LIN {X 0,Y 334.107,Z 246.869,A -85,B 0,C 180,E1 -14402.411,E2 -14402.411} C_VEL
LIN {X 0,Y 334.001,Z 246.88,A -85,B 0,C 180,E1 -14406.039,E2 -14406.039} C_VEL
LIN {X 0,Y 333.851,Z 246.902,A -85,B 0,C 180,E1 -14409.695,E2 -14409.695} C_VEL
LIN {X 0,Y 333.799,Z 246.904,A -85,B 0,C 180,E1 -14413.391,E2 -14413.391} C_VEL
LIN {X 0,Y 333.749,Z 246.913,A -85,B 0,C 180,E1 -14417.146,E2 -14417.146} C_VEL
LIN {X 0,Y 333.733,Z 246.914,A -85,B 0,C 180,E1 -14419.69,E2 -14419.69} C_VEL
LIN {X 0,Y 333.671,Z 246.922,A -85,B 0,C 180,E1 -14423.59,E2 -14423.59} C_VEL
LIN {X 0,Y 333.737,Z 246.913,A -85,B 0,C 180,E1 -14426.246,E2 -14426.246} C_VEL
LIN {X 0,Y 333.712,Z 246.915,A -85,B 0,C 180,E1 -14428.972,E2 -14428.972} C_VEL
LIN {X 0,Y 333.644,Z 246.924,A -85,B 0,C 180,E1 -14432.587,E2 -14432.587} C_VEL
LIN {X 0,Y 333.677,Z 246.921,A -85,B 0,C 180,E1 -14436.139,E2 -14436.139} C_VEL
LIN {X 0,Y 333.648,Z 246.924,A -85,B 0,C 180,E1 -14439.192,E2 -14439.192} C_VEL
LIN {X 0,Y 333.633,Z 246.926,A -85,B 0,C 180,E1 -14442.5,E2 -14442.5} C_VEL
LIN {X 0,Y 333.712,Z 246.938,A -85,B 0,C 180,E1 -14445.328,E2 -14445.328} C_VEL
LIN {X 0,Y 334.719,Z 252.739,A -85,B 0,C 180,E1 -14449.103,E2 -14449.103} C_VEL
LIN {X 0,Y 335.65,Z 258.414,A -85,B 0,C 180,E1 -14452.612,E2 -14452.612} C_VEL
LIN {X 0,Y 335.639,Z 262.053,A -85,B 0,C 180,E1 -14454.749,E2 -14454.749} C_VEL
LIN {X 0,Y 334.952,Z 267.23,A -85,B 0,C 180,E1 -14457.686,E2 -14457.686} C_VEL
LIN {X 0,Y 334.191,Z 273.317,A -85,B 0,C 180,E1 -14461.074,E2 -14461.074} C_VEL
LIN {X 0,Y 333.454,Z 280.637,A -85,B 0,C 180,E1 -14465.069,E2 -14465.069} C_VEL
LIN {X 0,Y 332.776,Z 289.063,A -85,B 0,C 180,E1 -14469.606,E2 -14469.606} C_VEL
LIN {X 0,Y 332.684,Z 290.253,A -85,B 0,C 180,E1 -14470.245,E2 -14470.245} C_VEL
LIN {X 0,Y 334.148,Z 304.974,A -85,B 0,C 180,E1 -14471.018,E2 -14471.018} C_VEL
LIN {X 0,Y 335.643,Z 318.794,A -85,B 0,C 180,E1 -14472.01,E2 -14472.01} C_VEL
LIN {X 0,Y 336.423,Z 328.102,A -85,B 0,C 180,E1 -14472.838,E2 -14472.838} C_VEL
LIN {X 0,Y 335.563,Z 339.641,A -85,B 0,C 180,E1 -14474.045,E2 -14474.045} C_VEL
LIN {X 0,Y 333.991,Z 358.219,A -85,B 0,C 180,E1 -14476.462,E2 -14476.462} C_VEL
LIN {X 0,Y 333.555,Z 364.929,A -85,B 0,C 180,E1 -14477.528,E2 -14477.528} C_VEL
LIN {X 0,Y 333.023,Z 371.307,A -85,B 0,C 180,E1 -14478.743,E2 -14478.743} C_VEL
LIN {X 0,Y 332.731,Z 376.622,A -85,B 0,C 180,E1 -14479.965,E2 -14479.965} C_VEL
LIN {X 0,Y 332.426,Z 382.036,A -85,B 0,C 180,E1 -14481.49,E2 -14481.49} C_VEL
LIN {X 0,Y 332.268,Z 385.533,A -85,B 0,C 180,E1 -14482.709,E2 -14482.709} C_VEL
LIN {X 0,Y 332.147,Z 389.249,A -85,B 0,C 180,E1 -14484.369,E2 -14484.369} C_VEL
LIN {X 0,Y 332.154,Z 390.661,A -85,B 0,C 180,E1 -14485.145,E2 -14485.145} C_VEL
LIN {X 0,Y 332.127,Z 392.341,A -85,B 0,C 180,E1 -14486.36,E2 -14486.36} C_VEL
LIN {X 0,Y 332.214,Z 393.428,A -85,B 0,C 180,E1 -14487.575,E2 -14487.575} C_VEL
LIN {X 0,Y 332.272,Z 394.91,A -85,B 0,C 180,E1 -14490,E2 -14490} C_VEL
LIN {X 0,Y 332.242,Z 395.234,A -85,B 0,C 180,E1 -14491.212,E2 -14491.212} C_VEL
LIN {X 0,Y 332.041,Z 394.613,A -85,B 0,C 180,E1 -14493.641,E2 -14493.641} C_VEL
LIN {X 0,Y 332.016,Z 392.694,A -85,B 0,C 180,E1 -14495.799,E2 -14495.799} C_VEL
LIN {X 0,Y 332.304,Z 389.55,A -85,B 0,C 180,E1 -14497.902,E2 -14497.902} C_VEL
LIN {X 0,Y 332.944,Z 384.242,A -85,B 0,C 180,E1 -14500.336,E2 -14500.336} C_VEL
LIN {X 0,Y 333.706,Z 379.024,A -85,B 0,C 180,E1 -14502.158,E2 -14502.158} C_VEL
LIN {X 0,Y 335.272,Z 371.438,A -85,B 0,C 180,E1 -14504.259,E2 -14504.259} C_VEL
LIN {X 0,Y 336.714,Z 362.936,A -85,B 0,C 180,E1 -14506.161,E2 -14506.161} C_VEL
LIN {X 0,Y 338.653,Z 353.757,A -85,B 0,C 180,E1 -14507.825,E2 -14507.825} C_VEL
LIN {X 0,Y 340.868,Z 342.995,A -85,B 0,C 180,E1 -14509.419,E2 -14509.419} C_VEL
LIN {X 0,Y 342.503,Z 333.768,A -85,B 0,C 180,E1 -14510.573,E2 -14510.573} C_VEL
LIN {X 0,Y 342.83,Z 323.695,A -85,B 0,C 180,E1 -14511.782,E2 -14511.782} C_VEL
LIN {X 0,Y 342.026,Z 313.427,A -85,B 0,C 180,E1 -14512.981,E2 -14512.981} C_VEL
LIN {X 0,Y 340.158,Z 302.986,A -85,B 0,C 180,E1 -14514.205,E2 -14514.205} C_VEL
LIN {X 0,Y 336.876,Z 291.319,A -85,B 0,C 180,E1 -14515.631,E2 -14515.631} C_VEL
LIN {X 0,Y 335.028,Z 286.128,A -85,B 0,C 180,E1 -14516.307,E2 -14516.307} C_VEL
LIN {X 0,Y 334.269,Z 282.995,A -85,B 0,C 180,E1 -14516.664,E2 -14516.664} C_VEL
LIN {X 0,Y 335.356,Z 276.756,A -85,B 0,C 180,E1 -14520.77,E2 -14520.77} C_VEL
LIN {X 0,Y 336.148,Z 273.348,A -85,B 0,C 180,E1 -14523.249,E2 -14523.249} C_VEL
LIN {X 0,Y 336.786,Z 270.249,A -85,B 0,C 180,E1 -14525.754,E2 -14525.754} C_VEL
LIN {X 0,Y 337.064,Z 268.24,A -85,B 0,C 180,E1 -14527.597,E2 -14527.597} C_VEL
LIN {X 0,Y 336.933,Z 265.791,A -85,B 0,C 180,E1 -14530.288,E2 -14530.288} C_VEL
LIN {X 0,Y 336.564,Z 263.455,A -85,B 0,C 180,E1 -14533.559,E2 -14533.559} C_VEL
LIN {X 0,Y 336.277,Z 261.677,A -85,B 0,C 180,E1 -14537.011,E2 -14537.011} C_VEL
LIN {X 0,Y 335.976,Z 260.544,A -85,B 0,C 180,E1 -14540.713,E2 -14540.713} C_VEL
LIN {X 0,Y 335.745,Z 260.144,A -85,B 0,C 180,E1 -14544.118,E2 -14544.118} C_VEL
LIN {X 0,Y 335.365,Z 260.286,A -85,B 0,C 180,E1 -14546.985,E2 -14546.985} C_VEL
LIN {X 0,Y 334.984,Z 260.763,A -85,B 0,C 180,E1 -14549.767,E2 -14549.767} C_VEL
LIN {X 0,Y 334.411,Z 261.974,A -85,B 0,C 180,E1 -14553.811,E2 -14553.811} C_VEL
LIN {X 0,Y 334.334,Z 262.309,A -85,B 0,C 180,E1 -14554.528,E2 -14554.528} C_VEL
LIN {X 0,Y 334.864,Z 264.05,A -85,B 0,C 180,E1 -14554.756,E2 -14554.756} C_VEL
LIN {X 0,Y 338.581,Z 270.778,A -85,B 0,C 180,E1 -14555.969,E2 -14555.969} C_VEL
LIN {X 0,Y 343.241,Z 281.46,A -85,B 0,C 180,E1 -14557.694,E2 -14557.694} C_VEL
LIN {X 0,Y 346.366,Z 292.219,A -85,B 0,C 180,E1 -14559.293,E2 -14559.293} C_VEL
LIN {X 0,Y 346.815,Z 295.222,A -85,B 0,C 180,E1 -14559.717,E2 -14559.717} C_VEL
LIN {X 0,Y 344.832,Z 306.353,A -85,B 0,C 180,E1 -14560.968,E2 -14560.968} C_VEL
LIN {X 0,Y 342.725,Z 316.647,A -85,B 0,C 180,E1 -14562.394,E2 -14562.394} C_VEL
LIN {X 0,Y 340.539,Z 326.819,A -85,B 0,C 180,E1 -14564.13,E2 -14564.13} C_VEL
LIN {X 0,Y 338.354,Z 336.288,A -85,B 0,C 180,E1 -14566.18,E2 -14566.18} C_VEL
LIN {X 0,Y 336.741,Z 342.83,A -85,B 0,C 180,E1 -14567.954,E2 -14567.954} C_VEL
LIN {X 0,Y 335.277,Z 349.062,A -85,B 0,C 180,E1 -14570.134,E2 -14570.134} C_VEL
LIN {X 0,Y 334.087,Z 353.412,A -85,B 0,C 180,E1 -14572.141,E2 -14572.141} C_VEL
LIN {X 0,Y 333.564,Z 356.202,A -85,B 0,C 180,E1 -14573.953,E2 -14573.953} C_VEL
LIN {X 0,Y 333.198,Z 357.575,A -85,B 0,C 180,E1 -14575.16,E2 -14575.16} C_VEL
LIN {X 0,Y 332.997,Z 358.506,A -85,B 0,C 180,E1 -14576.37,E2 -14576.37} C_VEL
LIN {X 0,Y 332.592,Z 359.055,A -85,B 0,C 180,E1 -14577.578,E2 -14577.578} C_VEL
LIN {X 0,Y 332.302,Z 358.959,A -85,B 0,C 180,E1 -14580,E2 -14580} C_VEL
LIN {X 0,Y 332.241,Z 358.27,A -85,B 0,C 180,E1 -14581.212,E2 -14581.212} C_VEL
LIN {X 0,Y 332.216,Z 357.176,A -85,B 0,C 180,E1 -14582.425,E2 -14582.425} C_VEL
LIN {X 0,Y 332.231,Z 355.68,A -85,B 0,C 180,E1 -14583.639,E2 -14583.639} C_VEL
LIN {X 0,Y 332.363,Z 352.595,A -85,B 0,C 180,E1 -14585.46,E2 -14585.46} C_VEL
LIN {X 0,Y 332.578,Z 348.448,A -85,B 0,C 180,E1 -14587.284,E2 -14587.284} C_VEL
LIN {X 0,Y 332.963,Z 342.109,A -85,B 0,C 180,E1 -14589.415,E2 -14589.415} C_VEL
LIN {X 0,Y 333.471,Z 335.212,A -85,B 0,C 180,E1 -14591.242,E2 -14591.242} C_VEL
LIN {X 0,Y 334.212,Z 326.729,A -85,B 0,C 180,E1 -14593.065,E2 -14593.065} C_VEL
LIN {X 0,Y 335.081,Z 316.348,A -85,B 0,C 180,E1 -14594.853,E2 -14594.853} C_VEL
LIN {X 0,Y 335.892,Z 305.186,A -85,B 0,C 180,E1 -14596.408,E2 -14596.408} C_VEL
LIN {X 0,Y 336.975,Z 292.951,A -85,B 0,C 180,E1 -14597.76,E2 -14597.76} C_VEL
LIN {X 0,Y 337.747,Z 281.884,A -85,B 0,C 180,E1 -14598.744,E2 -14598.744} C_VEL
LIN {X 0,Y 335.335,Z 269.091,A -85,B 0,C 180,E1 -14599.734,E2 -14599.734} C_VEL
LIN {X 0,Y 332.636,Z 255.172,A -85,B 0,C 180,E1 -14600.564,E2 -14600.564} C_VEL
LIN {X 0,Y 332.461,Z 254.001,A -85,B 0,C 180,E1 -14600.656,E2 -14600.656} C_VEL
LIN {X 0,Y 332.485,Z 249.793,A -85,B 0,C 180,E1 -14605.009,E2 -14605.009} C_VEL
LIN {X 0,Y 332.619,Z 247.259,A -85,B 0,C 180,E1 -14607.7,E2 -14607.7} C_VEL
LIN {X 0,Y 332.875,Z 247.018,A -85,B 0,C 180,E1 -14610.445,E2 -14610.445} C_VEL
LIN {X 0,Y 333.23,Z 246.978,A -85,B 0,C 180,E1 -14613.255,E2 -14613.255} C_VEL
LIN {X 0,Y 333.626,Z 246.926,A -85,B 0,C 180,E1 -14616.822,E2 -14616.822} C_VEL
LIN {X 0,Y 333.646,Z 246.927,A -85,B 0,C 180,E1 -14619.193,E2 -14619.193} C_VEL
LIN {X 0,Y 333.635,Z 246.924,A -85,B 0,C 180,E1 -14622.5,E2 -14622.5} C_VEL
LIN {X 0,Y 333.599,Z 246.927,A -85,B 0,C 180,E1 -14625.955,E2 -14625.955} C_VEL
LIN {X 0,Y 333.605,Z 246.929,A -85,B 0,C 180,E1 -14629.324,E2 -14629.324} C_VEL
LIN {X 0,Y 333.664,Z 246.922,A -85,B 0,C 180,E1 -14633.169,E2 -14633.169} C_VEL
LIN {X 0,Y 333.675,Z 246.919,A -85,B 0,C 180,E1 -14635.341,E2 -14635.341} C_VEL
LIN {X 0,Y 333.633,Z 246.925,A -85,B 0,C 180,E1 -14638.222,E2 -14638.222} C_VEL
LIN {X 0,Y 333.673,Z 246.92,A -85,B 0,C 180,E1 -14641.024,E2 -14641.024} C_VEL
LIN {X 0,Y 333.717,Z 246.913,A -85,B 0,C 180,E1 -14645.09,E2 -14645.09} C_VEL
LIN {X 0,Y 333.676,Z 246.918,A -85,B 0,C 180,E1 -14649.019,E2 -14649.019} C_VEL
LIN {X 0,Y 333.797,Z 246.903,A -85,B 0,C 180,E1 -14651.589,E2 -14651.589} C_VEL
LIN {X 0,Y 333.812,Z 246.902,A -85,B 0,C 180,E1 -14655.576,E2 -14655.576} C_VEL
LIN {X 0,Y 333.821,Z 246.9,A -85,B 0,C 180,E1 -14659.077,E2 -14659.077} C_VEL
LIN {X 0,Y 333.957,Z 246.883,A -85,B 0,C 180,E1 -14662.746,E2 -14662.746} C_VEL
LIN {X 0,Y 333.776,Z 246.906,A -85,B 0,C 180,E1 -14665.168,E2 -14665.168} C_VEL
LIN {X 0,Y 334.06,Z 246.874,A -85,B 0,C 180,E1 -14667.588,E2 -14667.588} C_VEL
LIN {X 0,Y 334.063,Z 246.871,A -85,B 0,C 180,E1 -14671.205,E2 -14671.205} C_VEL
LIN {X 0,Y 334.064,Z 246.87,A -85,B 0,C 180,E1 -14672.411,E2 -14672.411} C_VEL
LIN {X 0,Y 333.731,Z 247.126,A -85,B 0,C 180,E1 -14674.529,E2 -14674.529} C_VEL
LIN {X 0,Y 333.843,Z 251.062,A -85,B 0,C 180,E1 -14676.649,E2 -14676.649} C_VEL
LIN {X 0,Y 333.51,Z 259.079,A -85,B 0,C 180,E1 -14680.933,E2 -14680.933} C_VEL
LIN {X 0,Y 333.313,Z 266.04,A -85,B 0,C 180,E1 -14684.656,E2 -14684.656} C_VEL
LIN {X 0,Y 333.132,Z 273.18,A -85,B 0,C 180,E1 -14688.448,E2 -14688.448} C_VEL
LIN {X 0,Y 333.005,Z 277.43,A -85,B 0,C 180,E1 -14690.621,E2 -14690.621} C_VEL
LIN {X 0,Y 334.824,Z 287.032,A -85,B 0,C 180,E1 -14691.131,E2 -14691.131} C_VEL
LIN {X 0,Y 336.456,Z 296.89,A -85,B 0,C 180,E1 -14691.825,E2 -14691.825} C_VEL
LIN {X 0,Y 336.856,Z 299.779,A -85,B 0,C 180,E1 -14692.058,E2 -14692.058} C_VEL
LIN {X 0,Y 336.252,Z 309.946,A -85,B 0,C 180,E1 -14692.987,E2 -14692.987} C_VEL
LIN {X 0,Y 335.633,Z 318.187,A -85,B 0,C 180,E1 -14693.935,E2 -14693.935} C_VEL
LIN {X 0,Y 334.969,Z 326.014,A -85,B 0,C 180,E1 -14695.042,E2 -14695.042} C_VEL
LIN {X 0,Y 334.241,Z 334.509,A -85,B 0,C 180,E1 -14696.54,E2 -14696.54} C_VEL
LIN {X 0,Y 333.594,Z 341.051,A -85,B 0,C 180,E1 -14698.024,E2 -14698.024} C_VEL
LIN {X 0,Y 333.092,Z 346.387,A -85,B 0,C 180,E1 -14699.538,E2 -14699.538} C_VEL
LIN {X 0,Y 332.658,Z 350.895,A -85,B 0,C 180,E1 -14701.172,E2 -14701.172} C_VEL
LIN {X 0,Y 332.46,Z 353.233,A -85,B 0,C 180,E1 -14702.266,E2 -14702.266} C_VEL
LIN {X 0,Y 332.282,Z 355.148,A -85,B 0,C 180,E1 -14703.361,E2 -14703.361} C_VEL
LIN {X 0,Y 332.067,Z 356.989,A -85,B 0,C 180,E1 -14704.851,E2 -14704.851} C_VEL
LIN {X 0,Y 331.995,Z 358.079,A -85,B 0,C 180,E1 -14706.445,E2 -14706.445} C_VEL
LIN {X 0,Y 332.041,Z 358.213,A -85,B 0,C 180,E1 -14708.45,E2 -14708.45} C_VEL
LIN {X 0,Y 332.28,Z 357.086,A -85,B 0,C 180,E1 -14710.409,E2 -14710.409} C_VEL
LIN {X 0,Y 332.779,Z 354.245,A -85,B 0,C 180,E1 -14712.517,E2 -14712.517} C_VEL
LIN {X 0,Y 333.239,Z 350.815,A -85,B 0,C 180,E1 -14714.187,E2 -14714.187} C_VEL
LIN {X 0,Y 333.765,Z 346.626,A -85,B 0,C 180,E1 -14715.72,E2 -14715.72} C_VEL
LIN {X 0,Y 334.536,Z 340.977,A -85,B 0,C 180,E1 -14717.331,E2 -14717.331} C_VEL
LIN {X 0,Y 335.439,Z 333.566,A -85,B 0,C 180,E1 -14718.961,E2 -14718.961} C_VEL
LIN {X 0,Y 336.414,Z 325.791,A -85,B 0,C 180,E1 -14720.297,E2 -14720.297} C_VEL
LIN {X 0,Y 337.273,Z 317.796,A -85,B 0,C 180,E1 -14721.411,E2 -14721.411} C_VEL
LIN {X 0,Y 338.18,Z 307.72,A -85,B 0,C 180,E1 -14722.529,E2 -14722.529} C_VEL
LIN {X 0,Y 338.539,Z 302.937,A -85,B 0,C 180,E1 -14722.945,E2 -14722.945} C_VEL
LIN {X 0,Y 338.002,Z 300.173,A -85,B 0,C 180,E1 -14723.227,E2 -14723.227} C_VEL
LIN {X 0,Y 335.84,Z 296.788,A -85,B 0,C 180,E1 -14723.63,E2 -14723.63} C_VEL
LIN {X 0,Y 330.327,Z 290.415,A -85,B 0,C 180,E1 -14724.419,E2 -14724.419} C_VEL
LIN {X 0,Y 328.765,Z 287.073,A -85,B 0,C 180,E1 -14724.717,E2 -14724.717} C_VEL
LIN {X 0,Y 326.558,Z 278.694,A -85,B 0,C 180,E1 -14725.276,E2 -14725.276} C_VEL
LIN {X 0,Y 326.821,Z 271.194,A -85,B 0,C 180,E1 -14729.335,E2 -14729.335} C_VEL
LIN {X 0,Y 327.068,Z 265.376,A -85,B 0,C 180,E1 -14732.484,E2 -14732.484} C_VEL
LIN {X 0,Y 327.358,Z 258.958,A -85,B 0,C 180,E1 -14735.926,E2 -14735.926} C_VEL
LIN {X 0,Y 327.544,Z 254.11,A -85,B 0,C 180,E1 -14738.607,E2 -14738.607} C_VEL
LIN {X 0,Y 327.016,Z 249.609,A -85,B 0,C 180,E1 -14741.018,E2 -14741.018} C_VEL
LIN {X 0,Y 326.726,Z 247.788,A -85,B 0,C 180,E1 -14742.15,E2 -14742.15} C_VEL
LIN {X 0,Y 326.761,Z 247.784,A -85,B 0,C 180,E1 -14746.315,E2 -14746.315} C_VEL
LIN {X 0,Y 326.807,Z 247.78,A -85,B 0,C 180,E1 -14750.093,E2 -14750.093} C_VEL
LIN {X 0,Y 326.932,Z 247.762,A -85,B 0,C 180,E1 -14752.589,E2 -14752.589} C_VEL
LIN {X 0,Y 326.77,Z 247.783,A -85,B 0,C 180,E1 -14755.065,E2 -14755.065} C_VEL
LIN {X 0,Y 327.048,Z 247.747,A -85,B 0,C 180,E1 -14757.537,E2 -14757.537} C_VEL
LIN {X 0,Y 327.2,Z 247.728,A -85,B 0,C 180,E1 -14760,E2 -14760} C_VEL
LIN {X 0,Y 327.047,Z 247.749,A -85,B 0,C 180,E1 -14762.463,E2 -14762.463} C_VEL
LIN {X 0,Y 326.954,Z 247.757,A -85,B 0,C 180,E1 -14766.17,E2 -14766.17} C_VEL
LIN {X 0,Y 326.807,Z 247.778,A -85,B 0,C 180,E1 -14769.906,E2 -14769.906} C_VEL
LIN {X 0,Y 326.761,Z 247.78,A -85,B 0,C 180,E1 -14773.685,E2 -14773.685} C_VEL
LIN {X 0,Y 326.701,Z 247.791,A -85,B 0,C 180,E1 -14777.528,E2 -14777.528} C_VEL
LIN {X 0,Y 326.659,Z 247.797,A -85,B 0,C 180,E1 -14780.135,E2 -14780.135} C_VEL
LIN {X 0,Y 326.65,Z 247.794,A -85,B 0,C 180,E1 -14784.129,E2 -14784.129} C_VEL
LIN {X 0,Y 326.686,Z 247.788,A -85,B 0,C 180,E1 -14786.857,E2 -14786.857} C_VEL
LIN {X 0,Y 326.64,Z 247.798,A -85,B 0,C 180,E1 -14790.611,E2 -14790.611} C_VEL
LIN {X 0,Y 326.608,Z 247.801,A -85,B 0,C 180,E1 -14794.019,E2 -14794.019} C_VEL
LIN {X 0,Y 326.629,Z 247.796,A -85,B 0,C 180,E1 -14797.239,E2 -14797.239} C_VEL
LIN {X 0,Y 326.579,Z 247.806,A -85,B 0,C 180,E1 -14801.131,E2 -14801.131} C_VEL
LIN {X 0,Y 326.653,Z 247.934,A -85,B 0,C 180,E1 -14805.235,E2 -14805.235} C_VEL
LIN {X 0,Y 327.592,Z 253.087,A -85,B 0,C 180,E1 -14808.666,E2 -14808.666} C_VEL
LIN {X 0,Y 328.546,Z 258.835,A -85,B 0,C 180,E1 -14812.324,E2 -14812.324} C_VEL
LIN {X 0,Y 328.646,Z 262.186,A -85,B 0,C 180,E1 -14814.353,E2 -14814.353} C_VEL
LIN {X 0,Y 328.162,Z 266.11,A -85,B 0,C 180,E1 -14816.64,E2 -14816.64} C_VEL
LIN {X 0,Y 327.114,Z 273.906,A -85,B 0,C 180,E1 -14821.092,E2 -14821.092} C_VEL
LIN {X 0,Y 326.398,Z 280.406,A -85,B 0,C 180,E1 -14824.735,E2 -14824.735} C_VEL
LIN {X 0,Y 325.718,Z 288.366,A -85,B 0,C 180,E1 -14829.144,E2 -14829.144} C_VEL
LIN {X 0,Y 325.64,Z 289.929,A -85,B 0,C 180,E1 -14830.003,E2 -14830.003} C_VEL
LIN {X 0,Y 327.025,Z 304.811,A -85,B 0,C 180,E1 -14830.807,E2 -14830.807} C_VEL
LIN {X 0,Y 328.441,Z 317.82,A -85,B 0,C 180,E1 -14831.763,E2 -14831.763} C_VEL
LIN {X 0,Y 329.323,Z 328.91,A -85,B 0,C 180,E1 -14832.776,E2 -14832.776} C_VEL
LIN {X 0,Y 327.613,Z 350.293,A -85,B 0,C 180,E1 -14835.083,E2 -14835.083} C_VEL
LIN {X 0,Y 327.096,Z 358.256,A -85,B 0,C 180,E1 -14836.171,E2 -14836.171} C_VEL
LIN {X 0,Y 326.591,Z 364.889,A -85,B 0,C 180,E1 -14837.257,E2 -14837.257} C_VEL
LIN {X 0,Y 326.039,Z 371.198,A -85,B 0,C 180,E1 -14838.499,E2 -14838.499} C_VEL
LIN {X 0,Y 325.691,Z 376.456,A -85,B 0,C 180,E1 -14839.745,E2 -14839.745} C_VEL
LIN {X 0,Y 325.356,Z 381.819,A -85,B 0,C 180,E1 -14841.303,E2 -14841.303} C_VEL
LIN {X 0,Y 325.192,Z 385.278,A -85,B 0,C 180,E1 -14842.55,E2 -14842.55} C_VEL
LIN {X 0,Y 325.105,Z 388.379,A -85,B 0,C 180,E1 -14843.94,E2 -14843.94} C_VEL
LIN {X 0,Y 325.054,Z 390.343,A -85,B 0,C 180,E1 -14845.039,E2 -14845.039} C_VEL
LIN {X 0,Y 325.051,Z 392.016,A -85,B 0,C 180,E1 -14846.281,E2 -14846.281} C_VEL
LIN {X 0,Y 325.113,Z 393.084,A -85,B 0,C 180,E1 -14847.522,E2 -14847.522} C_VEL
LIN {X 0,Y 325.213,Z 394.338,A -85,B 0,C 180,E1 -14850,E2 -14850} C_VEL
LIN {X 0,Y 325.16,Z 394.757,A -85,B 0,C 180,E1 -14851.239,E2 -14851.239} C_VEL
LIN {X 0,Y 324.968,Z 394.709,A -85,B 0,C 180,E1 -14852.479,E2 -14852.479} C_VEL
LIN {X 0,Y 324.964,Z 394.256,A -85,B 0,C 180,E1 -14853.72,E2 -14853.72} C_VEL
LIN {X 0,Y 324.959,Z 392.143,A -85,B 0,C 180,E1 -14856.208,E2 -14856.208} C_VEL
LIN {X 0,Y 325.231,Z 389.447,A -85,B 0,C 180,E1 -14858.075,E2 -14858.075} C_VEL
LIN {X 0,Y 325.721,Z 385.776,A -85,B 0,C 180,E1 -14859.94,E2 -14859.94} C_VEL
LIN {X 0,Y 326.457,Z 381.087,A -85,B 0,C 180,E1 -14861.801,E2 -14861.801} C_VEL
LIN {X 0,Y 327.951,Z 374.197,A -85,B 0,C 180,E1 -14863.951,E2 -14863.951} C_VEL
LIN {X 0,Y 329.561,Z 365.556,A -85,B 0,C 180,E1 -14866.095,E2 -14866.095} C_VEL
LIN {X 0,Y 331.58,Z 356.505,A -85,B 0,C 180,E1 -14867.899,E2 -14867.899} C_VEL
LIN {X 0,Y 334.07,Z 345.476,A -85,B 0,C 180,E1 -14869.67,E2 -14869.67} C_VEL
LIN {X 0,Y 336.094,Z 335.617,A -85,B 0,C 180,E1 -14870.984,E2 -14870.984} C_VEL
LIN {X 0,Y 336.641,Z 327.06,A -85,B 0,C 180,E1 -14872.073,E2 -14872.073} C_VEL
LIN {X 0,Y 336.089,Z 316.381,A -85,B 0,C 180,E1 -14873.411,E2 -14873.411} C_VEL
LIN {X 0,Y 334.213,Z 304.829,A -85,B 0,C 180,E1 -14874.871,E2 -14874.871} C_VEL
LIN {X 0,Y 330.988,Z 292.612,A -85,B 0,C 180,E1 -14876.481,E2 -14876.481} C_VEL
LIN {X 0,Y 328.61,Z 286.055,A -85,B 0,C 180,E1 -14877.431,E2 -14877.431} C_VEL
LIN {X 0,Y 327.563,Z 282.454,A -85,B 0,C 180,E1 -14877.903,E2 -14877.903} C_VEL
LIN {X 0,Y 327.601,Z 281.842,A -85,B 0,C 180,E1 -14878.162,E2 -14878.162} C_VEL
LIN {X 0,Y 328.815,Z 275.97,A -85,B 0,C 180,E1 -14882.3,E2 -14882.3} C_VEL
LIN {X 0,Y 329.649,Z 272.408,A -85,B 0,C 180,E1 -14885.144,E2 -14885.144} C_VEL
LIN {X 0,Y 330.11,Z 269.322,A -85,B 0,C 180,E1 -14888.026,E2 -14888.026} C_VEL
LIN {X 0,Y 330.042,Z 267.601,A -85,B 0,C 180,E1 -14889.951,E2 -14889.951} C_VEL
LIN {X 0,Y 329.727,Z 265.367,A -85,B 0,C 180,E1 -14893.006,E2 -14893.006} C_VEL
LIN {X 0,Y 329.41,Z 263.477,A -85,B 0,C 180,E1 -14896.502,E2 -14896.502} C_VEL
LIN {X 0,Y 329.077,Z 262.224,A -85,B 0,C 180,E1 -14900.251,E2 -14900.251} C_VEL
LIN {X 0,Y 328.871,Z 261.739,A -85,B 0,C 180,E1 -14903.247,E2 -14903.247} C_VEL
LIN {X 0,Y 328.797,Z 261.657,A -85,B 0,C 180,E1 -14904.752,E2 -14904.752} C_VEL
LIN {X 0,Y 328.136,Z 262.06,A -85,B 0,C 180,E1 -14908.951,E2 -14908.951} C_VEL
LIN {X 0,Y 327.694,Z 262.742,A -85,B 0,C 180,E1 -14911.847,E2 -14911.847} C_VEL
LIN {X 0,Y 327.516,Z 263.246,A -85,B 0,C 180,E1 -14913.236,E2 -14913.236} C_VEL
LIN {X 0,Y 328.049,Z 264.951,A -85,B 0,C 180,E1 -14913.493,E2 -14913.493} C_VEL
LIN {X 0,Y 329.978,Z 267.913,A -85,B 0,C 180,E1 -14914.149,E2 -14914.149} C_VEL
LIN {X 0,Y 334.358,Z 276.867,A -85,B 0,C 180,E1 -14915.813,E2 -14915.813} C_VEL
LIN {X 0,Y 337.868,Z 285.506,A -85,B 0,C 180,E1 -14917.311,E2 -14917.311} C_VEL
LIN {X 0,Y 340.315,Z 294.398,A -85,B 0,C 180,E1 -14918.732,E2 -14918.732} C_VEL
LIN {X 0,Y 340.827,Z 297.077,A -85,B 0,C 180,E1 -14919.147,E2 -14919.147} C_VEL
LIN {X 0,Y 338.468,Z 309.183,A -85,B 0,C 180,E1 -14920.596,E2 -14920.596} C_VEL
LIN {X 0,Y 336.224,Z 319.075,A -85,B 0,C 180,E1 -14922.042,E2 -14922.042} C_VEL
LIN {X 0,Y 333.939,Z 328.778,A -85,B 0,C 180,E1 -14923.808,E2 -14923.808} C_VEL
LIN {X 0,Y 331.946,Z 336.742,A -85,B 0,C 180,E1 -14925.595,E2 -14925.595} C_VEL
LIN {X 0,Y 329.958,Z 344.203,A -85,B 0,C 180,E1 -14927.702,E2 -14927.702} C_VEL
LIN {X 0,Y 328.481,Z 349.925,A -85,B 0,C 180,E1 -14929.801,E2 -14929.801} C_VEL
LIN {X 0,Y 327.354,Z 353.281,A -85,B 0,C 180,E1 -14931.357,E2 -14931.357} C_VEL
LIN {X 0,Y 326.967,Z 355.352,A -85,B 0,C 180,E1 -14932.59,E2 -14932.59} C_VEL
LIN {X 0,Y 326.561,Z 357.032,A -85,B 0,C 180,E1 -14933.823,E2 -14933.823} C_VEL
LIN {X 0,Y 326.172,Z 358.284,A -85,B 0,C 180,E1 -14935.056,E2 -14935.056} C_VEL
LIN {X 0,Y 325.944,Z 359.122,A -85,B 0,C 180,E1 -14936.291,E2 -14936.291} C_VEL
LIN {X 0,Y 325.54,Z 359.597,A -85,B 0,C 180,E1 -14937.525,E2 -14937.525} C_VEL
LIN {X 0,Y 325.334,Z 359.673,A -85,B 0,C 180,E1 -14938.762,E2 -14938.762} C_VEL
LIN {X 0,Y 325.223,Z 359.308,A -85,B 0,C 180,E1 -14940,E2 -14940} C_VEL
LIN {X 0,Y 325.146,Z 358.539,A -85,B 0,C 180,E1 -14941.239,E2 -14941.239} C_VEL
LIN {X 0,Y 325.121,Z 357.376,A -85,B 0,C 180,E1 -14942.478,E2 -14942.478} C_VEL
LIN {X 0,Y 325.196,Z 354.818,A -85,B 0,C 180,E1 -14944.338,E2 -14944.338} C_VEL
LIN {X 0,Y 325.37,Z 350.642,A -85,B 0,C 180,E1 -14946.48,E2 -14946.48} C_VEL
LIN {X 0,Y 325.692,Z 344.743,A -85,B 0,C 180,E1 -14948.688,E2 -14948.688} C_VEL
LIN {X 0,Y 326.156,Z 338.394,A -85,B 0,C 180,E1 -14950.554,E2 -14950.554} C_VEL
LIN {X 0,Y 326.789,Z 330.55,A -85,B 0,C 180,E1 -14952.419,E2 -14952.419} C_VEL
LIN {X 0,Y 327.661,Z 320.786,A -85,B 0,C 180,E1 -14954.28,E2 -14954.28} C_VEL
LIN {X 0,Y 328.508,Z 310.171,A -85,B 0,C 180,E1 -14955.926,E2 -14955.926} C_VEL
LIN {X 0,Y 329.524,Z 298.513,A -85,B 0,C 180,E1 -14957.373,E2 -14957.373} C_VEL
LIN {X 0,Y 330.501,Z 286.156,A -85,B 0,C 180,E1 -14958.601,E2 -14958.601} C_VEL
LIN {X 0,Y 330.626,Z 282.261,A -85,B 0,C 180,E1 -14958.936,E2 -14958.936} C_VEL
LIN {X 0,Y 328.289,Z 269.759,A -85,B 0,C 180,E1 -14959.927,E2 -14959.927} C_VEL
LIN {X 0,Y 325.586,Z 255.785,A -85,B 0,C 180,E1 -14960.784,E2 -14960.784} C_VEL
LIN {X 0,Y 325.36,Z 254.38,A -85,B 0,C 180,E1 -14960.88,E2 -14960.88} C_VEL
LIN {X 0,Y 325.43,Z 250.536,A -85,B 0,C 180,E1 -14964.9,E2 -14964.9} C_VEL
LIN {X 0,Y 325.57,Z 247.936,A -85,B 0,C 180,E1 -14967.74,E2 -14967.74} C_VEL
LIN {X 0,Y 325.887,Z 247.891,A -85,B 0,C 180,E1 -14971.17,E2 -14971.17} C_VEL
LIN {X 0,Y 326.259,Z 247.842,A -85,B 0,C 180,E1 -14974.061,E2 -14974.061} C_VEL
LIN {X 0,Y 326.599,Z 247.805,A -85,B 0,C 180,E1 -14977.231,E2 -14977.231} C_VEL
LIN {X 0,Y 326.594,Z 247.8,A -85,B 0,C 180,E1 -14980.209,E2 -14980.209} C_VEL
LIN {X 0,Y 326.565,Z 247.805,A -85,B 0,C 180,E1 -14983.525,E2 -14983.525} C_VEL
LIN {X 0,Y 326.577,Z 247.807,A -85,B 0,C 180,E1 -14987.029,E2 -14987.029} C_VEL
LIN {X 0,Y 326.584,Z 247.802,A -85,B 0,C 180,E1 -14991.385,E2 -14991.385} C_VEL
LIN {X 0,Y 326.621,Z 247.801,A -85,B 0,C 180,E1 -14994.852,E2 -14994.852} C_VEL
LIN {X 0,Y 326.611,Z 247.798,A -85,B 0,C 180,E1 -14997.455,E2 -14997.455} C_VEL
LIN {X 0,Y 326.628,Z 247.799,A -85,B 0,C 180,E1 -15000.337,E2 -15000.337} C_VEL
LIN {X 0,Y 326.631,Z 247.796,A -85,B 0,C 180,E1 -15003.137,E2 -15003.137} C_VEL
LIN {X 0,Y 326.647,Z 247.795,A -85,B 0,C 180,E1 -15005.87,E2 -15005.87} C_VEL
LIN {X 0,Y 326.661,Z 247.793,A -85,B 0,C 180,E1 -15009.865,E2 -15009.865} C_VEL
LIN {X 0,Y 326.703,Z 247.79,A -85,B 0,C 180,E1 -15012.472,E2 -15012.472} C_VEL
LIN {X 0,Y 326.763,Z 247.783,A -85,B 0,C 180,E1 -15016.314,E2 -15016.314} C_VEL
LIN {X 0,Y 326.786,Z 247.781,A -85,B 0,C 180,E1 -15020.093,E2 -15020.093} C_VEL
LIN {X 0,Y 326.941,Z 247.762,A -85,B 0,C 180,E1 -15023.83,E2 -15023.83} C_VEL
LIN {X 0,Y 327.004,Z 247.752,A -85,B 0,C 180,E1 -15027.536,E2 -15027.536} C_VEL
LIN {X 0,Y 327.033,Z 247.747,A -85,B 0,C 180,E1 -15031.231,E2 -15031.231} C_VEL
LIN {X 0,Y 327.006,Z 247.749,A -85,B 0,C 180,E1 -15032.463,E2 -15032.463} C_VEL
LIN {X 0,Y 326.722,Z 247.916,A -85,B 0,C 180,E1 -15034.318,E2 -15034.318} C_VEL
LIN {X 0,Y 326.856,Z 251.304,A -85,B 0,C 180,E1 -15036.172,E2 -15036.172} C_VEL
LIN {X 0,Y 326.513,Z 259.405,A -85,B 0,C 180,E1 -15040.542,E2 -15040.542} C_VEL
LIN {X 0,Y 326.308,Z 266.27,A -85,B 0,C 180,E1 -15044.254,E2 -15044.254} C_VEL
LIN {X 0,Y 326.151,Z 272.419,A -85,B 0,C 180,E1 -15047.558,E2 -15047.558} C_VEL
LIN {X 0,Y 325.955,Z 277.542,A -85,B 0,C 180,E1 -15050.304,E2 -15050.304} C_VEL
LIN {X 0,Y 327.986,Z 288.464,A -85,B 0,C 180,E1 -15050.91,E2 -15050.91} C_VEL
LIN {X 0,Y 329.768,Z 299.521,A -85,B 0,C 180,E1 -15051.734,E2 -15051.734} C_VEL
LIN {X 0,Y 329.341,Z 309.936,A -85,B 0,C 180,E1 -15052.702,E2 -15052.702} C_VEL
LIN {X 0,Y 328.763,Z 317.51,A -85,B 0,C 180,E1 -15053.575,E2 -15053.575} C_VEL
LIN {X 0,Y 328.074,Z 325.427,A -85,B 0,C 180,E1 -15054.691,E2 -15054.691} C_VEL
LIN {X 0,Y 327.467,Z 332.258,A -85,B 0,C 180,E1 -15055.866,E2 -15055.866} C_VEL
LIN {X 0,Y 326.697,Z 340.162,A -85,B 0,C 180,E1 -15057.549,E2 -15057.549} C_VEL
LIN {X 0,Y 326.168,Z 345.447,A -85,B 0,C 180,E1 -15059,E2 -15059} C_VEL
LIN {X 0,Y 325.697,Z 350.365,A -85,B 0,C 180,E1 -15060.728,E2 -15060.728} C_VEL
LIN {X 0,Y 325.308,Z 354.496,A -85,B 0,C 180,E1 -15062.691,E2 -15062.691} C_VEL
LIN {X 0,Y 324.987,Z 357.277,A -85,B 0,C 180,E1 -15064.737,E2 -15064.737} C_VEL
LIN {X 0,Y 324.895,Z 358.569,A -85,B 0,C 180,E1 -15066.834,E2 -15066.834} C_VEL
LIN {X 0,Y 325.001,Z 358.531,A -85,B 0,C 180,E1 -15068.878,E2 -15068.878} C_VEL
LIN {X 0,Y 325.292,Z 357.162,A -85,B 0,C 180,E1 -15070.871,E2 -15070.871} C_VEL
LIN {X 0,Y 325.784,Z 354.422,A -85,B 0,C 180,E1 -15072.822,E2 -15072.822} C_VEL
LIN {X 0,Y 326.174,Z 351.78,A -85,B 0,C 180,E1 -15074.162,E2 -15074.162} C_VEL
LIN {X 0,Y 326.541,Z 349.139,A -85,B 0,C 180,E1 -15075.255,E2 -15075.255} C_VEL
LIN {X 0,Y 327.236,Z 343.974,A -85,B 0,C 180,E1 -15076.904,E2 -15076.904} C_VEL
LIN {X 0,Y 328.052,Z 338.119,A -85,B 0,C 180,E1 -15078.384,E2 -15078.384} C_VEL
LIN {X 0,Y 328.809,Z 332.293,A -85,B 0,C 180,E1 -15079.589,E2 -15079.589} C_VEL
LIN {X 0,Y 329.751,Z 324.972,A -85,B 0,C 180,E1 -15080.829,E2 -15080.829} C_VEL
LIN {X 0,Y 330.73,Z 316.002,A -85,B 0,C 180,E1 -15082.058,E2 -15082.058} C_VEL
LIN {X 0,Y 331.675,Z 305.867,A -85,B 0,C 180,E1 -15083.111,E2 -15083.111} C_VEL
LIN {X 0,Y 331.657,Z 302.602,A -85,B 0,C 180,E1 -15083.417,E2 -15083.417} C_VEL
LIN {X 0,Y 330.049,Z 292.897,A -85,B 0,C 180,E1 -15084.287,E2 -15084.287} C_VEL
LIN {X 0,Y 328.765,Z 287.073,A -85,B 0,C 180,E1 -15084.717,E2 -15084.717} C_VEL
LIN {X 0,Y 327.267,Z 283.819,A -85,B 0,C 180,E1 -15085.055,E2 -15085.055} C_VEL
LIN {X 0,Y 325.114,Z 281.299,A -85,B 0,C 180,E1 -15085.49,E2 -15085.49} C_VEL
LIN {X 0,Y 322.139,Z 278.779,A -85,B 0,C 180,E1 -15086.192,E2 -15086.192} C_VEL
LIN {X 0,Y 320.025,Z 276.803,A -85,B 0,C 180,E1 -15087.033,E2 -15087.033} C_VEL
LIN {X 0,Y 319.703,Z 275.921,A -85,B 0,C 180,E1 -15087.494,E2 -15087.494} C_VEL
LIN {X 0,Y 320.025,Z 268.715,A -85,B 0,C 180,E1 -15091.454,E2 -15091.454} C_VEL
LIN {X 0,Y 320.429,Z 260.334,A -85,B 0,C 180,E1 -15096.061,E2 -15096.061} C_VEL
LIN {X 0,Y 320.602,Z 255.302,A -85,B 0,C 180,E1 -15098.795,E2 -15098.795} C_VEL
LIN {X 0,Y 320.007,Z 250.468,A -85,B 0,C 180,E1 -15101.489,E2 -15101.489} C_VEL
LIN {X 0,Y 319.669,Z 248.668,A -85,B 0,C 180,E1 -15102.569,E2 -15102.569} C_VEL
LIN {X 0,Y 319.739,Z 248.66,A -85,B 0,C 180,E1 -15106.008,E2 -15106.008} C_VEL
LIN {X 0,Y 319.754,Z 248.658,A -85,B 0,C 180,E1 -15109.873,E2 -15109.873} C_VEL
LIN {X 0,Y 319.892,Z 248.639,A -85,B 0,C 180,E1 -15112.425,E2 -15112.425} C_VEL
LIN {X 0,Y 319.738,Z 248.659,A -85,B 0,C 180,E1 -15114.956,E2 -15114.956} C_VEL
LIN {X 0,Y 319.991,Z 248.626,A -85,B 0,C 180,E1 -15117.482,E2 -15117.482} C_VEL
LIN {X 0,Y 320.151,Z 248.606,A -85,B 0,C 180,E1 -15120,E2 -15120} C_VEL
LIN {X 0,Y 319.991,Z 248.628,A -85,B 0,C 180,E1 -15122.517,E2 -15122.517} C_VEL
LIN {X 0,Y 319.911,Z 248.635,A -85,B 0,C 180,E1 -15126.306,E2 -15126.306} C_VEL
LIN {X 0,Y 319.754,Z 248.656,A -85,B 0,C 180,E1 -15130.127,E2 -15130.127} C_VEL
LIN {X 0,Y 319.733,Z 248.659,A -85,B 0,C 180,E1 -15134.724,E2 -15134.724} C_VEL
LIN {X 0,Y 319.69,Z 248.661,A -85,B 0,C 180,E1 -15139.037,E2 -15139.037} C_VEL
LIN {X 0,Y 319.561,Z 248.68,A -85,B 0,C 180,E1 -15143.32,E2 -15143.32} C_VEL
LIN {X 0,Y 319.636,Z 248.67,A -85,B 0,C 180,E1 -15146.088,E2 -15146.088} C_VEL
LIN {X 0,Y 319.591,Z 248.674,A -85,B 0,C 180,E1 -15148.933,E2 -15148.933} C_VEL
LIN {X 0,Y 319.533,Z 248.68,A -85,B 0,C 180,E1 -15151.862,E2 -15151.862} C_VEL
LIN {X 0,Y 319.581,Z 248.676,A -85,B 0,C 180,E1 -15155.543,E2 -15155.543} C_VEL
LIN {X 0,Y 319.574,Z 248.677,A -85,B 0,C 180,E1 -15158.008,E2 -15158.008} C_VEL
LIN {X 0,Y 319.527,Z 248.683,A -85,B 0,C 180,E1 -15161.597,E2 -15161.597} C_VEL
LIN {X 0,Y 319.586,Z 248.723,A -85,B 0,C 180,E1 -15165.013,E2 -15165.013} C_VEL
LIN {X 0,Y 320.629,Z 254.41,A -85,B 0,C 180,E1 -15168.884,E2 -15168.884} C_VEL
LIN {X 0,Y 321.486,Z 259.61,A -85,B 0,C 180,E1 -15172.258,E2 -15172.258} C_VEL
LIN {X 0,Y 321.531,Z 263.491,A -85,B 0,C 180,E1 -15174.658,E2 -15174.658} C_VEL
LIN {X 0,Y 320.817,Z 268.331,A -85,B 0,C 180,E1 -15177.54,E2 -15177.54} C_VEL
LIN {X 0,Y 319.919,Z 275.105,A -85,B 0,C 180,E1 -15181.489,E2 -15181.489} C_VEL
LIN {X 0,Y 319.222,Z 281.695,A -85,B 0,C 180,E1 -15185.272,E2 -15185.272} C_VEL
LIN {X 0,Y 318.57,Z 289.445,A -85,B 0,C 180,E1 -15189.668,E2 -15189.668} C_VEL
LIN {X 0,Y 318.67,Z 291.065,A -85,B 0,C 180,E1 -15189.843,E2 -15189.843} C_VEL
LIN {X 0,Y 319.921,Z 304.515,A -85,B 0,C 180,E1 -15190.594,E2 -15190.594} C_VEL
LIN {X 0,Y 321.423,Z 318.77,A -85,B 0,C 180,E1 -15191.681,E2 -15191.681} C_VEL
LIN {X 0,Y 322.239,Z 329.575,A -85,B 0,C 180,E1 -15192.713,E2 -15192.713} C_VEL
LIN {X 0,Y 321.493,Z 342.367,A -85,B 0,C 180,E1 -15193.849,E2 -15193.849} C_VEL
LIN {X 0,Y 320.633,Z 351.599,A -85,B 0,C 180,E1 -15194.913,E2 -15194.913} C_VEL
LIN {X 0,Y 320.092,Z 359.307,A -85,B 0,C 180,E1 -15196.024,E2 -15196.024} C_VEL
LIN {X 0,Y 319.386,Z 368.223,A -85,B 0,C 180,E1 -15197.611,E2 -15197.611} C_VEL
LIN {X 0,Y 318.732,Z 375.124,A -85,B 0,C 180,E1 -15199.198,E2 -15199.198} C_VEL
LIN {X 0,Y 318.405,Z 379.684,A -85,B 0,C 180,E1 -15200.471,E2 -15200.471} C_VEL
LIN {X 0,Y 318.196,Z 383.489,A -85,B 0,C 180,E1 -15201.746,E2 -15201.746} C_VEL
LIN {X 0,Y 318.019,Z 387.826,A -85,B 0,C 180,E1 -15203.656,E2 -15203.656} C_VEL
LIN {X 0,Y 317.962,Z 390.032,A -85,B 0,C 180,E1 -15204.928,E2 -15204.928} C_VEL
LIN {X 0,Y 317.975,Z 391.69,A -85,B 0,C 180,E1 -15206.198,E2 -15206.198} C_VEL
LIN {X 0,Y 318.017,Z 392.741,A -85,B 0,C 180,E1 -15207.467,E2 -15207.467} C_VEL
LIN {X 0,Y 318.156,Z 393.756,A -85,B 0,C 180,E1 -15210,E2 -15210} C_VEL
LIN {X 0,Y 318.08,Z 394.231,A -85,B 0,C 180,E1 -15211.266,E2 -15211.266} C_VEL
LIN {X 0,Y 317.881,Z 394.286,A -85,B 0,C 180,E1 -15212.535,E2 -15212.535} C_VEL
LIN {X 0,Y 317.887,Z 393.902,A -85,B 0,C 180,E1 -15213.803,E2 -15213.803} C_VEL
LIN {X 0,Y 317.888,Z 391.912,A -85,B 0,C 180,E1 -15216.347,E2 -15216.347} C_VEL
LIN {X 0,Y 318.18,Z 389.347,A -85,B 0,C 180,E1 -15218.255,E2 -15218.255} C_VEL
LIN {X 0,Y 318.709,Z 385.82,A -85,B 0,C 180,E1 -15220.161,E2 -15220.161} C_VEL
LIN {X 0,Y 319.481,Z 381.296,A -85,B 0,C 180,E1 -15222.063,E2 -15222.063} C_VEL
LIN {X 0,Y 321.086,Z 374.627,A -85,B 0,C 180,E1 -15224.256,E2 -15224.256} C_VEL
LIN {X 0,Y 322.786,Z 366.27,A -85,B 0,C 180,E1 -15226.443,E2 -15226.443} C_VEL
LIN {X 0,Y 324.904,Z 357.514,A -85,B 0,C 180,E1 -15228.28,E2 -15228.28} C_VEL
LIN {X 0,Y 327.519,Z 346.939,A -85,B 0,C 180,E1 -15230.08,E2 -15230.08} C_VEL
LIN {X 0,Y 329.814,Z 336.363,A -85,B 0,C 180,E1 -15231.567,E2 -15231.567} C_VEL
LIN {X 0,Y 330.44,Z 327.784,A -85,B 0,C 180,E1 -15232.725,E2 -15232.725} C_VEL
LIN {X 0,Y 330.026,Z 317.934,A -85,B 0,C 180,E1 -15234.042,E2 -15234.042} C_VEL
LIN {X 0,Y 328.341,Z 306.735,A -85,B 0,C 180,E1 -15235.564,E2 -15235.564} C_VEL
LIN {X 0,Y 325.617,Z 295.705,A -85,B 0,C 180,E1 -15237.135,E2 -15237.135} C_VEL
LIN {X 0,Y 324.035,Z 290.79,A -85,B 0,C 180,E1 -15237.893,E2 -15237.893} C_VEL
LIN {X 0,Y 322.85,Z 286.772,A -85,B 0,C 180,E1 -15238.49,E2 -15238.49} C_VEL
LIN {X 0,Y 321.265,Z 283.289,A -85,B 0,C 180,E1 -15239.119,E2 -15239.119} C_VEL
LIN {X 0,Y 320.907,Z 281.273,A -85,B 0,C 180,E1 -15239.392,E2 -15239.392} C_VEL
LIN {X 0,Y 322.064,Z 276.346,A -85,B 0,C 180,E1 -15243.062,E2 -15243.062} C_VEL
LIN {X 0,Y 322.953,Z 272.494,A -85,B 0,C 180,E1 -15246.372,E2 -15246.372} C_VEL
LIN {X 0,Y 323.114,Z 269.852,A -85,B 0,C 180,E1 -15249.108,E2 -15249.108} C_VEL
LIN {X 0,Y 322.874,Z 267.428,A -85,B 0,C 180,E1 -15252.262,E2 -15252.262} C_VEL
LIN {X 0,Y 322.531,Z 265.309,A -85,B 0,C 180,E1 -15255.979,E2 -15255.979} C_VEL
LIN {X 0,Y 322.218,Z 264.119,A -85,B 0,C 180,E1 -15259.13,E2 -15259.13} C_VEL
LIN {X 0,Y 322.016,Z 263.415,A -85,B 0,C 180,E1 -15262.331,E2 -15262.331} C_VEL
LIN {X 0,Y 321.742,Z 263.21,A -85,B 0,C 180,E1 -15265.394,E2 -15265.394} C_VEL
LIN {X 0,Y 321.245,Z 263.491,A -85,B 0,C 180,E1 -15268.564,E2 -15268.564} C_VEL
LIN {X 0,Y 320.796,Z 264.324,A -85,B 0,C 180,E1 -15271.788,E2 -15271.788} C_VEL
LIN {X 0,Y 322.035,Z 267.308,A -85,B 0,C 180,E1 -15272.372,E2 -15272.372} C_VEL
LIN {X 0,Y 323.559,Z 269.476,A -85,B 0,C 180,E1 -15272.945,E2 -15272.945} C_VEL
LIN {X 0,Y 327.614,Z 277.129,A -85,B 0,C 180,E1 -15274.593,E2 -15274.593} C_VEL
LIN {X 0,Y 332.017,Z 288.046,A -85,B 0,C 180,E1 -15276.656,E2 -15276.656} C_VEL
LIN {X 0,Y 334.4,Z 297.023,A -85,B 0,C 180,E1 -15278.205,E2 -15278.205} C_VEL
LIN {X 0,Y 334.833,Z 299.527,A -85,B 0,C 180,E1 -15278.62,E2 -15278.62} C_VEL
LIN {X 0,Y 332.367,Z 311.043,A -85,B 0,C 180,E1 -15280.064,E2 -15280.064} C_VEL
LIN {X 0,Y 329.764,Z 321.483,A -85,B 0,C 180,E1 -15281.678,E2 -15281.678} C_VEL
LIN {X 0,Y 327.375,Z 330.808,A -85,B 0,C 180,E1 -15283.474,E2 -15283.474} C_VEL
LIN {X 0,Y 325.269,Z 338.46,A -85,B 0,C 180,E1 -15285.293,E2 -15285.293} C_VEL
LIN {X 0,Y 323.163,Z 345.623,A -85,B 0,C 180,E1 -15287.439,E2 -15287.439} C_VEL
LIN {X 0,Y 321.719,Z 350.777,A -85,B 0,C 180,E1 -15289.433,E2 -15289.433} C_VEL
LIN {X 0,Y 320.425,Z 354.313,A -85,B 0,C 180,E1 -15291.168,E2 -15291.168} C_VEL
LIN {X 0,Y 319.992,Z 356.291,A -85,B 0,C 180,E1 -15292.428,E2 -15292.428} C_VEL
LIN {X 0,Y 319.561,Z 357.835,A -85,B 0,C 180,E1 -15293.687,E2 -15293.687} C_VEL
LIN {X 0,Y 318.894,Z 359.746,A -85,B 0,C 180,E1 -15296.209,E2 -15296.209} C_VEL
LIN {X 0,Y 318.489,Z 360.141,A -85,B 0,C 180,E1 -15297.471,E2 -15297.471} C_VEL
LIN {X 0,Y 318.258,Z 360.093,A -85,B 0,C 180,E1 -15298.735,E2 -15298.735} C_VEL
LIN {X 0,Y 318.131,Z 359.641,A -85,B 0,C 180,E1 -15300,E2 -15300} C_VEL
LIN {X 0,Y 318.05,Z 358.8,A -85,B 0,C 180,E1 -15301.266,E2 -15301.266} C_VEL
LIN {X 0,Y 318.03,Z 357.556,A -85,B 0,C 180,E1 -15302.533,E2 -15302.533} C_VEL
LIN {X 0,Y 318.114,Z 354.86,A -85,B 0,C 180,E1 -15304.435,E2 -15304.435} C_VEL
LIN {X 0,Y 318.348,Z 349.796,A -85,B 0,C 180,E1 -15306.911,E2 -15306.911} C_VEL
LIN {X 0,Y 318.635,Z 344.42,A -85,B 0,C 180,E1 -15308.882,E2 -15308.882} C_VEL
LIN {X 0,Y 319.121,Z 337.892,A -85,B 0,C 180,E1 -15310.789,E2 -15310.789} C_VEL
LIN {X 0,Y 319.829,Z 329.781,A -85,B 0,C 180,E1 -15312.694,E2 -15312.694} C_VEL
LIN {X 0,Y 320.737,Z 319.81,A -85,B 0,C 180,E1 -15314.595,E2 -15314.595} C_VEL
LIN {X 0,Y 321.554,Z 309.345,A -85,B 0,C 180,E1 -15316.205,E2 -15316.205} C_VEL
LIN {X 0,Y 322.55,Z 298.243,A -85,B 0,C 180,E1 -15317.597,E2 -15317.597} C_VEL
LIN {X 0,Y 323.415,Z 287.486,A -85,B 0,C 180,E1 -15318.695,E2 -15318.695} C_VEL
LIN {X 0,Y 323.502,Z 282.589,A -85,B 0,C 180,E1 -15319.13,E2 -15319.13} C_VEL
LIN {X 0,Y 321.18,Z 270.124,A -85,B 0,C 180,E1 -15320.142,E2 -15320.142} C_VEL
LIN {X 0,Y 318.385,Z 255.609,A -85,B 0,C 180,E1 -15321.047,E2 -15321.047} C_VEL
LIN {X 0,Y 318.285,Z 254.75,A -85,B 0,C 180,E1 -15321.112,E2 -15321.112} C_VEL
LIN {X 0,Y 318.379,Z 250.917,A -85,B 0,C 180,E1 -15325.169,E2 -15325.169} C_VEL
LIN {X 0,Y 318.507,Z 248.816,A -85,B 0,C 180,E1 -15327.605,E2 -15327.605} C_VEL
LIN {X 0,Y 318.796,Z 248.772,A -85,B 0,C 180,E1 -15330.708,E2 -15330.708} C_VEL
LIN {X 0,Y 319.146,Z 248.733,A -85,B 0,C 180,E1 -15333.404,E2 -15333.404} C_VEL
LIN {X 0,Y 319.48,Z 248.686,A -85,B 0,C 180,E1 -15336.438,E2 -15336.438} C_VEL
LIN {X 0,Y 319.562,Z 248.677,A -85,B 0,C 180,E1 -15339.669,E2 -15339.669} C_VEL
LIN {X 0,Y 319.525,Z 248.683,A -85,B 0,C 180,E1 -15343.461,E2 -15343.461} C_VEL
LIN {X 0,Y 319.555,Z 248.682,A -85,B 0,C 180,E1 -15347.016,E2 -15347.016} C_VEL
LIN {X 0,Y 319.548,Z 248.679,A -85,B 0,C 180,E1 -15350.37,E2 -15350.37} C_VEL
LIN {X 0,Y 319.581,Z 248.676,A -85,B 0,C 180,E1 -15354.457,E2 -15354.457} C_VEL
LIN {X 0,Y 319.528,Z 248.682,A -85,B 0,C 180,E1 -15358.137,E2 -15358.137} C_VEL
LIN {X 0,Y 319.597,Z 248.672,A -85,B 0,C 180,E1 -15361.596,E2 -15361.596} C_VEL
LIN {X 0,Y 319.587,Z 248.673,A -85,B 0,C 180,E1 -15365.302,E2 -15365.302} C_VEL
LIN {X 0,Y 319.605,Z 248.671,A -85,B 0,C 180,E1 -15369.4,E2 -15369.4} C_VEL
LIN {X 0,Y 319.662,Z 248.667,A -85,B 0,C 180,E1 -15372.073,E2 -15372.073} C_VEL
LIN {X 0,Y 319.736,Z 248.659,A -85,B 0,C 180,E1 -15376.008,E2 -15376.008} C_VEL
LIN {X 0,Y 319.739,Z 248.658,A -85,B 0,C 180,E1 -15379.872,E2 -15379.872} C_VEL
LIN {X 0,Y 319.899,Z 248.638,A -85,B 0,C 180,E1 -15383.693,E2 -15383.693} C_VEL
LIN {X 0,Y 320.012,Z 248.62,A -85,B 0,C 180,E1 -15388.741,E2 -15388.741} C_VEL
LIN {X 0,Y 319.951,Z 248.628,A -85,B 0,C 180,E1 -15392.518,E2 -15392.518} C_VEL
LIN {X 0,Y 319.683,Z 248.713,A -85,B 0,C 180,E1 -15394.097,E2 -15394.097} C_VEL
LIN {X 0,Y 319.834,Z 252.728,A -85,B 0,C 180,E1 -15396.308,E2 -15396.308} C_VEL
LIN {X 0,Y 319.484,Z 260.936,A -85,B 0,C 180,E1 -15400.777,E2 -15400.777} C_VEL
LIN {X 0,Y 319.263,Z 267.564,A -85,B 0,C 180,E1 -15404.399,E2 -15404.399} C_VEL
LIN {X 0,Y 319.074,Z 274.087,A -85,B 0,C 180,E1 -15407.961,E2 -15407.961} C_VEL
LIN {X 0,Y 318.936,Z 278.049,A -85,B 0,C 180,E1 -15410.014,E2 -15410.014} C_VEL
LIN {X 0,Y 320.834,Z 287.834,A -85,B 0,C 180,E1 -15410.559,E2 -15410.559} C_VEL
LIN {X 0,Y 322.36,Z 297.274,A -85,B 0,C 180,E1 -15411.251,E2 -15411.251} C_VEL
LIN {X 0,Y 322.905,Z 302.59,A -85,B 0,C 180,E1 -15411.716,E2 -15411.716} C_VEL
LIN {X 0,Y 322.289,Z 311.637,A -85,B 0,C 180,E1 -15412.603,E2 -15412.603} C_VEL
LIN {X 0,Y 321.605,Z 319.937,A -85,B 0,C 180,E1 -15413.62,E2 -15413.62} C_VEL
LIN {X 0,Y 320.878,Z 328.597,A -85,B 0,C 180,E1 -15414.937,E2 -15414.937} C_VEL
LIN {X 0,Y 320.118,Z 336.121,A -85,B 0,C 180,E1 -15416.396,E2 -15416.396} C_VEL
LIN {X 0,Y 319.462,Z 342.365,A -85,B 0,C 180,E1 -15417.904,E2 -15417.904} C_VEL
LIN {X 0,Y 318.984,Z 347.217,A -85,B 0,C 180,E1 -15419.355,E2 -15419.355} C_VEL
LIN {X 0,Y 318.475,Z 352.229,A -85,B 0,C 180,E1 -15421.276,E2 -15421.276} C_VEL
LIN {X 0,Y 318.167,Z 355.352,A -85,B 0,C 180,E1 -15422.924,E2 -15422.924} C_VEL
LIN {X 0,Y 317.871,Z 357.942,A -85,B 0,C 180,E1 -15425.109,E2 -15425.109} C_VEL
LIN {X 0,Y 317.812,Z 359.058,A -85,B 0,C 180,E1 -15427.241,E2 -15427.241} C_VEL
LIN {X 0,Y 317.964,Z 358.82,A -85,B 0,C 180,E1 -15429.32,E2 -15429.32} C_VEL
LIN {X 0,Y 318.357,Z 357.005,A -85,B 0,C 180,E1 -15431.474,E2 -15431.474} C_VEL
LIN {X 0,Y 318.79,Z 354.647,A -85,B 0,C 180,E1 -15433.112,E2 -15433.112} C_VEL
LIN {X 0,Y 319.291,Z 351.27,A -85,B 0,C 180,E1 -15434.778,E2 -15434.778} C_VEL
LIN {X 0,Y 320.122,Z 345.722,A -85,B 0,C 180,E1 -15436.799,E2 -15436.799} C_VEL
LIN {X 0,Y 321.105,Z 339.087,A -85,B 0,C 180,E1 -15438.562,E2 -15438.562} C_VEL
LIN {X 0,Y 321.907,Z 333.184,A -85,B 0,C 180,E1 -15439.83,E2 -15439.83} C_VEL
LIN {X 0,Y 322.883,Z 326.102,A -85,B 0,C 180,E1 -15441.075,E2 -15441.075} C_VEL
LIN {X 0,Y 323.913,Z 317.212,A -85,B 0,C 180,E1 -15442.343,E2 -15442.343} C_VEL
LIN {X 0,Y 324.971,Z 306.629,A -85,B 0,C 180,E1 -15443.491,E2 -15443.491} C_VEL
LIN {X 0,Y 324.738,Z 302.245,A -85,B 0,C 180,E1 -15443.928,E2 -15443.928} C_VEL
LIN {X 0,Y 322.63,Z 290.711,A -85,B 0,C 180,E1 -15444.946,E2 -15444.946} C_VEL
LIN {X 0,Y 320.132,Z 281.264,A -85,B 0,C 180,E1 -15445.624,E2 -15445.624} C_VEL
LIN {X 0,Y 319.569,Z 279.023,A -85,B 0,C 180,E1 -15445.793,E2 -15445.793} C_VEL
LIN {X 0,Y 319.703,Z 275.921,A -85,B 0,C 180,E1 -15447.494,E2 -15447.494} C_VEL
LIN {X 0,Y 319.131,Z 274.224,A -85,B 0,C 180,E1 -15448.502,E2 -15448.502} C_VEL
LIN {X 0,Y 316.497,Z 271.771,A -85,B 0,C 180,E1 -15450.165,E2 -15450.165} C_VEL
LIN {X 0,Y 314.236,Z 269.807,A -85,B 0,C 180,E1 -15451.514,E2 -15451.514} C_VEL
LIN {X 0,Y 313.259,Z 268.166,A -85,B 0,C 180,E1 -15452.548,E2 -15452.548} C_VEL
LIN {X 0,Y 313.177,Z 267.571,A -85,B 0,C 180,E1 -15452.895,E2 -15452.895} C_VEL
LIN {X 0,Y 313.551,Z 260.676,A -85,B 0,C 180,E1 -15456.778,E2 -15456.778} C_VEL
LIN {X 0,Y 313.649,Z 256.524,A -85,B 0,C 180,E1 -15458.991,E2 -15458.991} C_VEL
LIN {X 0,Y 313.067,Z 251.843,A -85,B 0,C 180,E1 -15461.682,E2 -15461.682} C_VEL
LIN {X 0,Y 312.615,Z 249.545,A -85,B 0,C 180,E1 -15463.175,E2 -15463.175} C_VEL
LIN {X 0,Y 312.702,Z 249.536,A -85,B 0,C 180,E1 -15465.686,E2 -15465.686} C_VEL
LIN {X 0,Y 312.7,Z 249.537,A -85,B 0,C 180,E1 -15469.642,E2 -15469.642} C_VEL
LIN {X 0,Y 312.836,Z 249.519,A -85,B 0,C 180,E1 -15472.253,E2 -15472.253} C_VEL
LIN {X 0,Y 312.707,Z 249.535,A -85,B 0,C 180,E1 -15474.842,E2 -15474.842} C_VEL
LIN {X 0,Y 312.991,Z 249.5,A -85,B 0,C 180,E1 -15478.713,E2 -15478.713} C_VEL
LIN {X 0,Y 312.991,Z 249.498,A -85,B 0,C 180,E1 -15481.287,E2 -15481.287} C_VEL
LIN {X 0,Y 312.708,Z 249.534,A -85,B 0,C 180,E1 -15485.158,E2 -15485.158} C_VEL
LIN {X 0,Y 312.819,Z 249.52,A -85,B 0,C 180,E1 -15487.747,E2 -15487.747} C_VEL
LIN {X 0,Y 312.671,Z 249.537,A -85,B 0,C 180,E1 -15491.671,E2 -15491.671} C_VEL
LIN {X 0,Y 312.702,Z 249.534,A -85,B 0,C 180,E1 -15494.888,E2 -15494.888} C_VEL
LIN {X 0,Y 312.63,Z 249.541,A -85,B 0,C 180,E1 -15499.236,E2 -15499.236} C_VEL
LIN {X 0,Y 312.527,Z 249.558,A -85,B 0,C 180,E1 -15502.78,E2 -15502.78} C_VEL
LIN {X 0,Y 312.604,Z 249.547,A -85,B 0,C 180,E1 -15505.935,E2 -15505.935} C_VEL
LIN {X 0,Y 312.546,Z 249.55,A -85,B 0,C 180,E1 -15509.65,E2 -15509.65} C_VEL
LIN {X 0,Y 312.52,Z 249.556,A -85,B 0,C 180,E1 -15513.689,E2 -15513.689} C_VEL
LIN {X 0,Y 312.527,Z 249.553,A -85,B 0,C 180,E1 -15517.385,E2 -15517.385} C_VEL
LIN {X 0,Y 312.491,Z 249.562,A -85,B 0,C 180,E1 -15520.709,E2 -15520.709} C_VEL
LIN {X 0,Y 312.552,Z 249.604,A -85,B 0,C 180,E1 -15524.87,E2 -15524.87} C_VEL
LIN {X 0,Y 313.553,Z 254.999,A -85,B 0,C 180,E1 -15528.631,E2 -15528.631} C_VEL
LIN {X 0,Y 314.441,Z 260.382,A -85,B 0,C 180,E1 -15532.209,E2 -15532.209} C_VEL
LIN {X 0,Y 314.494,Z 263.965,A -85,B 0,C 180,E1 -15534.478,E2 -15534.478} C_VEL
LIN {X 0,Y 313.765,Z 268.889,A -85,B 0,C 180,E1 -15537.481,E2 -15537.481} C_VEL
LIN {X 0,Y 312.904,Z 275.026,A -85,B 0,C 180,E1 -15541.159,E2 -15541.159} C_VEL
LIN {X 0,Y 312.213,Z 280.981,A -85,B 0,C 180,E1 -15544.679,E2 -15544.679} C_VEL
LIN {X 0,Y 311.574,Z 288.421,A -85,B 0,C 180,E1 -15548.931,E2 -15548.931} C_VEL
LIN {X 0,Y 311.897,Z 294.181,A -85,B 0,C 180,E1 -15549.773,E2 -15549.773} C_VEL
LIN {X 0,Y 313.309,Z 308.811,A -85,B 0,C 180,E1 -15550.706,E2 -15550.706} C_VEL
LIN {X 0,Y 314.642,Z 321.672,A -85,B 0,C 180,E1 -15551.707,E2 -15551.707} C_VEL
LIN {X 0,Y 315.459,Z 331.022,A -85,B 0,C 180,E1 -15552.413,E2 -15552.413} C_VEL
LIN {X 0,Y 314.813,Z 340.955,A -85,B 0,C 180,E1 -15553.296,E2 -15553.296} C_VEL
LIN {X 0,Y 313.922,Z 350.598,A -85,B 0,C 180,E1 -15554.416,E2 -15554.416} C_VEL
LIN {X 0,Y 313.398,Z 357.492,A -85,B 0,C 180,E1 -15555.407,E2 -15555.407} C_VEL
LIN {X 0,Y 312.872,Z 363.157,A -85,B 0,C 180,E1 -15556.358,E2 -15556.358} C_VEL
LIN {X 0,Y 312.29,Z 369.605,A -85,B 0,C 180,E1 -15557.655,E2 -15557.655} C_VEL
LIN {X 0,Y 311.721,Z 374.984,A -85,B 0,C 180,E1 -15558.952,E2 -15558.952} C_VEL
LIN {X 0,Y 311.363,Z 379.493,A -85,B 0,C 180,E1 -15560.254,E2 -15560.254} C_VEL
LIN {X 0,Y 311.035,Z 384.814,A -85,B 0,C 180,E1 -15562.208,E2 -15562.208} C_VEL
LIN {X 0,Y 310.923,Z 388.494,A -85,B 0,C 180,E1 -15564.023,E2 -15564.023} C_VEL
LIN {X 0,Y 310.878,Z 391.363,A -85,B 0,C 180,E1 -15566.111,E2 -15566.111} C_VEL
LIN {X 0,Y 310.925,Z 392.405,A -85,B 0,C 180,E1 -15567.409,E2 -15567.409} C_VEL
LIN {X 0,Y 311.099,Z 393.166,A -85,B 0,C 180,E1 -15570,E2 -15570} C_VEL
LIN {X 0,Y 311.002,Z 393.696,A -85,B 0,C 180,E1 -15571.295,E2 -15571.295} C_VEL
LIN {X 0,Y 310.79,Z 393.538,A -85,B 0,C 180,E1 -15573.89,E2 -15573.89} C_VEL
LIN {X 0,Y 310.755,Z 392.442,A -85,B 0,C 180,E1 -15575.674,E2 -15575.674} C_VEL
LIN {X 0,Y 311.004,Z 390.175,A -85,B 0,C 180,E1 -15577.793,E2 -15577.793} C_VEL
LIN {X 0,Y 311.443,Z 387.12,A -85,B 0,C 180,E1 -15579.744,E2 -15579.744} C_VEL
LIN {X 0,Y 312.204,Z 383.091,A -85,B 0,C 180,E1 -15581.689,E2 -15581.689} C_VEL
LIN {X 0,Y 313.4,Z 378.028,A -85,B 0,C 180,E1 -15583.619,E2 -15583.619} C_VEL
LIN {X 0,Y 314.952,Z 371.838,A -85,B 0,C 180,E1 -15585.532,E2 -15585.532} C_VEL
LIN {X 0,Y 316.621,Z 364.713,A -85,B 0,C 180,E1 -15587.356,E2 -15587.356} C_VEL
LIN {X 0,Y 319.135,Z 355.419,A -85,B 0,C 180,E1 -15589.289,E2 -15589.289} C_VEL
LIN {X 0,Y 321.957,Z 344.565,A -85,B 0,C 180,E1 -15591.112,E2 -15591.112} C_VEL
LIN {X 0,Y 323.614,Z 337.249,A -85,B 0,C 180,E1 -15592.169,E2 -15592.169} C_VEL
LIN {X 0,Y 324.301,Z 329.597,A -85,B 0,C 180,E1 -15593.263,E2 -15593.263} C_VEL
LIN {X 0,Y 324.015,Z 319.069,A -85,B 0,C 180,E1 -15594.768,E2 -15594.768} C_VEL
LIN {X 0,Y 322.448,Z 307.817,A -85,B 0,C 180,E1 -15596.414,E2 -15596.414} C_VEL
LIN {X 0,Y 319.407,Z 295.547,A -85,B 0,C 180,E1 -15598.342,E2 -15598.342} C_VEL
LIN {X 0,Y 317.793,Z 290.472,A -85,B 0,C 180,E1 -15599.21,E2 -15599.21} C_VEL
LIN {X 0,Y 316.408,Z 285.98,A -85,B 0,C 180,E1 -15599.973,E2 -15599.973} C_VEL
LIN {X 0,Y 314.775,Z 282.388,A -85,B 0,C 180,E1 -15600.716,E2 -15600.716} C_VEL
LIN {X 0,Y 314.431,Z 280.274,A -85,B 0,C 180,E1 -15601.066,E2 -15601.066} C_VEL
LIN {X 0,Y 315.535,Z 276.013,A -85,B 0,C 180,E1 -15604.501,E2 -15604.501} C_VEL
LIN {X 0,Y 316.041,Z 273.429,A -85,B 0,C 180,E1 -15606.9,E2 -15606.9} C_VEL
LIN {X 0,Y 316.19,Z 271.533,A -85,B 0,C 180,E1 -15608.927,E2 -15608.927} C_VEL
LIN {X 0,Y 315.99,Z 269.281,A -85,B 0,C 180,E1 -15611.855,E2 -15611.855} C_VEL
LIN {X 0,Y 315.657,Z 267.174,A -85,B 0,C 180,E1 -15615.437,E2 -15615.437} C_VEL
LIN {X 0,Y 315.415,Z 266.058,A -85,B 0,C 180,E1 -15618.052,E2 -15618.052} C_VEL
LIN {X 0,Y 315.158,Z 265.16,A -85,B 0,C 180,E1 -15621.362,E2 -15621.362} C_VEL
LIN {X 0,Y 314.905,Z 264.784,A -85,B 0,C 180,E1 -15624.531,E2 -15624.531} C_VEL
LIN {X 0,Y 314.449,Z 264.878,A -85,B 0,C 180,E1 -15627.561,E2 -15627.561} C_VEL
LIN {X 0,Y 314.081,Z 265.324,A -85,B 0,C 180,E1 -15630.076,E2 -15630.076} C_VEL
LIN {X 0,Y 314.98,Z 267.777,A -85,B 0,C 180,E1 -15630.602,E2 -15630.602} C_VEL
LIN {X 0,Y 316.581,Z 269.717,A -85,B 0,C 180,E1 -15631.269,E2 -15631.269} C_VEL
LIN {X 0,Y 318.216,Z 273.017,A -85,B 0,C 180,E1 -15632.06,E2 -15632.06} C_VEL
LIN {X 0,Y 319.215,Z 274.365,A -85,B 0,C 180,E1 -15632.461,E2 -15632.461} C_VEL
LIN {X 0,Y 323.443,Z 283.296,A -85,B 0,C 180,E1 -15634.473,E2 -15634.473} C_VEL
LIN {X 0,Y 326.858,Z 292.653,A -85,B 0,C 180,E1 -15636.356,E2 -15636.356} C_VEL
LIN {X 0,Y 328.856,Z 301.64,A -85,B 0,C 180,E1 -15638.003,E2 -15638.003} C_VEL
LIN {X 0,Y 326.289,Z 313,A -85,B 0,C 180,E1 -15639.512,E2 -15639.512} C_VEL
LIN {X 0,Y 323.33,Z 323.949,A -85,B 0,C 180,E1 -15641.3,E2 -15641.3} C_VEL
LIN {X 0,Y 320.828,Z 332.843,A -85,B 0,C 180,E1 -15643.127,E2 -15643.127} C_VEL
LIN {X 0,Y 318.283,Z 341.272,A -85,B 0,C 180,E1 -15645.29,E2 -15645.29} C_VEL
LIN {X 0,Y 316.391,Z 347.086,A -85,B 0,C 180,E1 -15647.166,E2 -15647.166} C_VEL
LIN {X 0,Y 314.923,Z 351.775,A -85,B 0,C 180,E1 -15649.094,E2 -15649.094} C_VEL
LIN {X 0,Y 313.5,Z 355.371,A -85,B 0,C 180,E1 -15650.972,E2 -15650.972} C_VEL
LIN {X 0,Y 312.564,Z 358.638,A -85,B 0,C 180,E1 -15653.545,E2 -15653.545} C_VEL
LIN {X 0,Y 311.847,Z 360.373,A -85,B 0,C 180,E1 -15656.123,E2 -15656.123} C_VEL
LIN {X 0,Y 311.44,Z 360.635,A -85,B 0,C 180,E1 -15657.413,E2 -15657.413} C_VEL
LIN {X 0,Y 311.038,Z 359.968,A -85,B 0,C 180,E1 -15660,E2 -15660} C_VEL
LIN {X 0,Y 310.954,Z 359.042,A -85,B 0,C 180,E1 -15661.295,E2 -15661.295} C_VEL
LIN {X 0,Y 310.943,Z 357.665,A -85,B 0,C 180,E1 -15662.591,E2 -15662.591} C_VEL
LIN {X 0,Y 311.035,Z 354.828,A -85,B 0,C 180,E1 -15664.536,E2 -15664.536} C_VEL
LIN {X 0,Y 311.189,Z 350.963,A -85,B 0,C 180,E1 -15666.484,E2 -15666.484} C_VEL
LIN {X 0,Y 311.457,Z 345.955,A -85,B 0,C 180,E1 -15668.434,E2 -15668.434} C_VEL
LIN {X 0,Y 312.007,Z 338.516,A -85,B 0,C 180,E1 -15670.71,E2 -15670.71} C_VEL
LIN {X 0,Y 312.681,Z 330.469,A -85,B 0,C 180,E1 -15672.659,E2 -15672.659} C_VEL
LIN {X 0,Y 313.609,Z 320.572,A -85,B 0,C 180,E1 -15674.603,E2 -15674.603} C_VEL
LIN {X 0,Y 314.403,Z 310.765,A -85,B 0,C 180,E1 -15676.171,E2 -15676.171} C_VEL
LIN {X 0,Y 315.435,Z 299.204,A -85,B 0,C 180,E1 -15677.672,E2 -15677.672} C_VEL
LIN {X 0,Y 316.459,Z 286.888,A -85,B 0,C 180,E1 -15678.953,E2 -15678.953} C_VEL
LIN {X 0,Y 316.42,Z 283.198,A -85,B 0,C 180,E1 -15679.293,E2 -15679.293} C_VEL
LIN {X 0,Y 314.1,Z 270.669,A -85,B 0,C 180,E1 -15680.338,E2 -15680.338} C_VEL
LIN {X 0,Y 311.354,Z 256.216,A -85,B 0,C 180,E1 -15681.27,E2 -15681.27} C_VEL
LIN {X 0,Y 311.202,Z 255.144,A -85,B 0,C 180,E1 -15681.326,E2 -15681.326} C_VEL
LIN {X 0,Y 311.302,Z 251.299,A -85,B 0,C 180,E1 -15685.437,E2 -15685.437} C_VEL
LIN {X 0,Y 311.358,Z 250.024,A -85,B 0,C 180,E1 -15686.836,E2 -15686.836} C_VEL
LIN {X 0,Y 311.506,Z 249.685,A -85,B 0,C 180,E1 -15688.369,E2 -15688.369} C_VEL
LIN {X 0,Y 311.99,Z 249.62,A -85,B 0,C 180,E1 -15692.727,E2 -15692.727} C_VEL
LIN {X 0,Y 312.408,Z 249.568,A -85,B 0,C 180,E1 -15695.916,E2 -15695.916} C_VEL
LIN {X 0,Y 312.495,Z 249.56,A -85,B 0,C 180,E1 -15699.03,E2 -15699.03} C_VEL
LIN {X 0,Y 312.493,Z 249.557,A -85,B 0,C 180,E1 -15702.432,E2 -15702.432} C_VEL
LIN {X 0,Y 312.461,Z 249.561,A -85,B 0,C 180,E1 -15706.035,E2 -15706.035} C_VEL
LIN {X 0,Y 312.458,Z 249.561,A -85,B 0,C 180,E1 -15709.885,E2 -15709.885} C_VEL
LIN {X 0,Y 312.536,Z 249.552,A -85,B 0,C 180,E1 -15714.051,E2 -15714.051} C_VEL
LIN {X 0,Y 312.505,Z 249.556,A -85,B 0,C 180,E1 -15717.333,E2 -15717.333} C_VEL
LIN {X 0,Y 312.527,Z 249.553,A -85,B 0,C 180,E1 -15721.285,E2 -15721.285} C_VEL
LIN {X 0,Y 312.558,Z 249.552,A -85,B 0,C 180,E1 -15724.708,E2 -15724.708} C_VEL
LIN {X 0,Y 312.567,Z 249.547,A -85,B 0,C 180,E1 -15727.527,E2 -15727.527} C_VEL
LIN {X 0,Y 312.642,Z 249.539,A -85,B 0,C 180,E1 -15731.656,E2 -15731.656} C_VEL
LIN {X 0,Y 312.697,Z 249.533,A -85,B 0,C 180,E1 -15735.686,E2 -15735.686} C_VEL
LIN {X 0,Y 312.689,Z 249.535,A -85,B 0,C 180,E1 -15739.641,E2 -15739.641} C_VEL
LIN {X 0,Y 312.798,Z 249.522,A -85,B 0,C 180,E1 -15742.252,E2 -15742.252} C_VEL
LIN {X 0,Y 312.686,Z 249.533,A -85,B 0,C 180,E1 -15744.842,E2 -15744.842} C_VEL
LIN {X 0,Y 312.979,Z 249.497,A -85,B 0,C 180,E1 -15748.713,E2 -15748.713} C_VEL
LIN {X 0,Y 312.97,Z 249.5,A -85,B 0,C 180,E1 -15751.287,E2 -15751.287} C_VEL
LIN {X 0,Y 312.657,Z 249.654,A -85,B 0,C 180,E1 -15753.947,E2 -15753.947} C_VEL
LIN {X 0,Y 312.812,Z 254.137,A -85,B 0,C 180,E1 -15756.45,E2 -15756.45} C_VEL
LIN {X 0,Y 312.447,Z 262.459,A -85,B 0,C 180,E1 -15761.022,E2 -15761.022} C_VEL
LIN {X 0,Y 312.175,Z 269.695,A -85,B 0,C 180,E1 -15765.005,E2 -15765.005} C_VEL
LIN {X 0,Y 311.979,Z 276.734,A -85,B 0,C 180,E1 -15768.889,E2 -15768.889} C_VEL
LIN {X 0,Y 311.899,Z 278.342,A -85,B 0,C 180,E1 -15769.69,E2 -15769.69} C_VEL
LIN {X 0,Y 313.702,Z 287.934,A -85,B 0,C 180,E1 -15770.234,E2 -15770.234} C_VEL
LIN {X 0,Y 315.228,Z 296.838,A -85,B 0,C 180,E1 -15770.899,E2 -15770.899} C_VEL
LIN {X 0,Y 315.949,Z 302.085,A -85,B 0,C 180,E1 -15771.361,E2 -15771.361} C_VEL
LIN {X 0,Y 315.423,Z 311.173,A -85,B 0,C 180,E1 -15772.258,E2 -15772.258} C_VEL
LIN {X 0,Y 314.717,Z 319.641,A -85,B 0,C 180,E1 -15773.3,E2 -15773.3} C_VEL
LIN {X 0,Y 313.911,Z 328.439,A -85,B 0,C 180,E1 -15774.644,E2 -15774.644} C_VEL
LIN {X 0,Y 313.159,Z 336.131,A -85,B 0,C 180,E1 -15776.143,E2 -15776.143} C_VEL
LIN {X 0,Y 312.556,Z 341.599,A -85,B 0,C 180,E1 -15777.449,E2 -15777.449} C_VEL
LIN {X 0,Y 311.953,Z 347.182,A -85,B 0,C 180,E1 -15779.109,E2 -15779.109} C_VEL
LIN {X 0,Y 311.463,Z 352.034,A -85,B 0,C 180,E1 -15780.968,E2 -15780.968} C_VEL
LIN {X 0,Y 311.098,Z 355.624,A -85,B 0,C 180,E1 -15782.832,E2 -15782.832} C_VEL
LIN {X 0,Y 310.854,Z 357.708,A -85,B 0,C 180,E1 -15784.417,E2 -15784.417} C_VEL
LIN {X 0,Y 310.742,Z 359.009,A -85,B 0,C 180,E1 -15786.018,E2 -15786.018} C_VEL
LIN {X 0,Y 310.746,Z 359.543,A -85,B 0,C 180,E1 -15787.666,E2 -15787.666} C_VEL
LIN {X 0,Y 310.957,Z 358.99,A -85,B 0,C 180,E1 -15789.785,E2 -15789.785} C_VEL
LIN {X 0,Y 311.154,Z 358.199,A -85,B 0,C 180,E1 -15790.921,E2 -15790.921} C_VEL
LIN {X 0,Y 311.579,Z 356.256,A -85,B 0,C 180,E1 -15792.585,E2 -15792.585} C_VEL
LIN {X 0,Y 312.06,Z 353.335,A -85,B 0,C 180,E1 -15794.28,E2 -15794.28} C_VEL
LIN {X 0,Y 312.682,Z 349.283,A -85,B 0,C 180,E1 -15795.993,E2 -15795.993} C_VEL
LIN {X 0,Y 313.569,Z 343.843,A -85,B 0,C 180,E1 -15797.748,E2 -15797.748} C_VEL
LIN {X 0,Y 314.285,Z 339.046,A -85,B 0,C 180,E1 -15799,E2 -15799} C_VEL
LIN {X 0,Y 315.245,Z 332.849,A -85,B 0,C 180,E1 -15800.331,E2 -15800.331} C_VEL
LIN {X 0,Y 316.158,Z 326.215,A -85,B 0,C 180,E1 -15801.506,E2 -15801.506} C_VEL
LIN {X 0,Y 317.335,Z 316.694,A -85,B 0,C 180,E1 -15802.872,E2 -15802.872} C_VEL
LIN {X 0,Y 318.356,Z 306.209,A -85,B 0,C 180,E1 -15804.001,E2 -15804.001} C_VEL
LIN {X 0,Y 317.156,Z 298.108,A -85,B 0,C 180,E1 -15804.82,E2 -15804.82} C_VEL
LIN {X 0,Y 315.246,Z 289.051,A -85,B 0,C 180,E1 -15805.596,E2 -15805.596} C_VEL
LIN {X 0,Y 312.609,Z 279.452,A -85,B 0,C 180,E1 -15806.287,E2 -15806.287} C_VEL
LIN {X 0,Y 312.895,Z 273.423,A -85,B 0,C 180,E1 -15809.643,E2 -15809.643} C_VEL
LIN {X 0,Y 313.177,Z 267.571,A -85,B 0,C 180,E1 -15812.895,E2 -15812.895} C_VEL
LIN {X 0,Y 312.538,Z 265.915,A -85,B 0,C 180,E1 -15813.925,E2 -15813.925} C_VEL
LIN {X 0,Y 309.866,Z 263.54,A -85,B 0,C 180,E1 -15815.626,E2 -15815.626} C_VEL
LIN {X 0,Y 307.656,Z 261.527,A -85,B 0,C 180,E1 -15817.004,E2 -15817.004} C_VEL
LIN {X 0,Y 306.772,Z 259.803,A -85,B 0,C 180,E1 -15818.056,E2 -15818.056} C_VEL
LIN {X 0,Y 306.732,Z 259.176,A -85,B 0,C 180,E1 -15818.409,E2 -15818.409} C_VEL
LIN {X 0,Y 306.435,Z 255.286,A -85,B 0,C 180,E1 -15820.645,E2 -15820.645} C_VEL
LIN {X 0,Y 305.601,Z 250.419,A -85,B 0,C 180,E1 -15823.809,E2 -15823.809} C_VEL
LIN {X 0,Y 305.593,Z 250.418,A -85,B 0,C 180,E1 -15826.704,E2 -15826.704} C_VEL
LIN {X 0,Y 305.788,Z 250.396,A -85,B 0,C 180,E1 -15831.22,E2 -15831.22} C_VEL
LIN {X 0,Y 305.802,Z 250.395,A -85,B 0,C 180,E1 -15833.401,E2 -15833.401} C_VEL
LIN {X 0,Y 305.886,Z 250.383,A -85,B 0,C 180,E1 -15837.366,E2 -15837.366} C_VEL
LIN {X 0,Y 306.056,Z 250.362,A -85,B 0,C 180,E1 -15840,E2 -15840} C_VEL
LIN {X 0,Y 305.886,Z 250.385,A -85,B 0,C 180,E1 -15842.634,E2 -15842.634} C_VEL
LIN {X 0,Y 305.8,Z 250.394,A -85,B 0,C 180,E1 -15846.598,E2 -15846.598} C_VEL
LIN {X 0,Y 305.699,Z 250.406,A -85,B 0,C 180,E1 -15849.261,E2 -15849.261} C_VEL
LIN {X 0,Y 305.591,Z 250.417,A -85,B 0,C 180,E1 -15853.296,E2 -15853.296} C_VEL
LIN {X 0,Y 305.596,Z 250.415,A -85,B 0,C 180,E1 -15856.02,E2 -15856.02} C_VEL
LIN {X 0,Y 305.577,Z 250.421,A -85,B 0,C 180,E1 -15859.444,E2 -15859.444} C_VEL
LIN {X 0,Y 305.487,Z 250.433,A -85,B 0,C 180,E1 -15863.039,E2 -15863.039} C_VEL
LIN {X 0,Y 305.549,Z 250.423,A -85,B 0,C 180,E1 -15866.227,E2 -15866.227} C_VEL
LIN {X 0,Y 305.497,Z 250.429,A -85,B 0,C 180,E1 -15869.05,E2 -15869.05} C_VEL
LIN {X 0,Y 305.466,Z 250.436,A -85,B 0,C 180,E1 -15873.517,E2 -15873.517} C_VEL
LIN {X 0,Y 305.476,Z 250.432,A -85,B 0,C 180,E1 -15876.739,E2 -15876.739} C_VEL
LIN {X 0,Y 305.455,Z 250.437,A -85,B 0,C 180,E1 -15880.6,E2 -15880.6} C_VEL
LIN {X 0,Y 305.554,Z 250.564,A -85,B 0,C 180,E1 -15884.797,E2 -15884.797} C_VEL
LIN {X 0,Y 306.642,Z 256.679,A -85,B 0,C 180,E1 -15889.142,E2 -15889.142} C_VEL
LIN {X 0,Y 307.311,Z 260.689,A -85,B 0,C 180,E1 -15891.868,E2 -15891.868} C_VEL
LIN {X 0,Y 307.505,Z 263.235,A -85,B 0,C 180,E1 -15893.542,E2 -15893.542} C_VEL
LIN {X 0,Y 307.263,Z 266.206,A -85,B 0,C 180,E1 -15895.429,E2 -15895.429} C_VEL
LIN {X 0,Y 306.167,Z 273.04,A -85,B 0,C 180,E1 -15899.668,E2 -15899.668} C_VEL
LIN {X 0,Y 305.258,Z 280.254,A -85,B 0,C 180,E1 -15904.059,E2 -15904.059} C_VEL
LIN {X 0,Y 304.593,Z 287.063,A -85,B 0,C 180,E1 -15908.075,E2 -15908.075} C_VEL
LIN {X 0,Y 305.222,Z 294.527,A -85,B 0,C 180,E1 -15909.267,E2 -15909.267} C_VEL
LIN {X 0,Y 305.176,Z 298.519,A -85,B 0,C 180,E1 -15909.816,E2 -15909.816} C_VEL
LIN {X 0,Y 306.209,Z 308.858,A -85,B 0,C 180,E1 -15910.462,E2 -15910.462} C_VEL
LIN {X 0,Y 307.517,Z 318.477,A -85,B 0,C 180,E1 -15911.006,E2 -15911.006} C_VEL
LIN {X 0,Y 308.565,Z 328.44,A -85,B 0,C 180,E1 -15911.749,E2 -15911.749} C_VEL
LIN {X 0,Y 308.649,Z 332.687,A -85,B 0,C 180,E1 -15912.098,E2 -15912.098} C_VEL
LIN {X 0,Y 308.009,Z 341.443,A -85,B 0,C 180,E1 -15912.933,E2 -15912.933} C_VEL
LIN {X 0,Y 307.093,Z 350.807,A -85,B 0,C 180,E1 -15914.06,E2 -15914.06} C_VEL
LIN {X 0,Y 306.504,Z 357.753,A -85,B 0,C 180,E1 -15915.097,E2 -15915.097} C_VEL
LIN {X 0,Y 305.794,Z 364.877,A -85,B 0,C 180,E1 -15916.375,E2 -15916.375} C_VEL
LIN {X 0,Y 304.949,Z 372.401,A -85,B 0,C 180,E1 -15918.029,E2 -15918.029} C_VEL
LIN {X 0,Y 304.341,Z 379.331,A -85,B 0,C 180,E1 -15920.027,E2 -15920.027} C_VEL
LIN {X 0,Y 303.985,Z 384.596,A -85,B 0,C 180,E1 -15922.027,E2 -15922.027} C_VEL
LIN {X 0,Y 303.839,Z 388.534,A -85,B 0,C 180,E1 -15924.054,E2 -15924.054} C_VEL
LIN {X 0,Y 303.786,Z 391.03,A -85,B 0,C 180,E1 -15926.02,E2 -15926.02} C_VEL
LIN {X 0,Y 303.835,Z 392.066,A -85,B 0,C 180,E1 -15927.349,E2 -15927.349} C_VEL
LIN {X 0,Y 303.927,Z 392.528,A -85,B 0,C 180,E1 -15928.675,E2 -15928.675} C_VEL
LIN {X 0,Y 304.044,Z 392.554,A -85,B 0,C 180,E1 -15930,E2 -15930} C_VEL
LIN {X 0,Y 303.926,Z 393.156,A -85,B 0,C 180,E1 -15931.325,E2 -15931.325} C_VEL
LIN {X 0,Y 303.697,Z 393.126,A -85,B 0,C 180,E1 -15933.981,E2 -15933.981} C_VEL
LIN {X 0,Y 303.66,Z 392.314,A -85,B 0,C 180,E1 -15935.612,E2 -15935.612} C_VEL
LIN {X 0,Y 303.94,Z 390.045,A -85,B 0,C 180,E1 -15937.975,E2 -15937.975} C_VEL
LIN {X 0,Y 304.674,Z 385.975,A -85,B 0,C 180,E1 -15940.634,E2 -15940.634} C_VEL
LIN {X 0,Y 305.582,Z 381.782,A -85,B 0,C 180,E1 -15942.621,E2 -15942.621} C_VEL
LIN {X 0,Y 307.129,Z 376.543,A -85,B 0,C 180,E1 -15944.579,E2 -15944.579} C_VEL
LIN {X 0,Y 308.98,Z 369.029,A -85,B 0,C 180,E1 -15946.859,E2 -15946.859} C_VEL
LIN {X 0,Y 311.636,Z 359.696,A -85,B 0,C 180,E1 -15949.087,E2 -15949.087} C_VEL
LIN {X 0,Y 314.488,Z 349.939,A -85,B 0,C 180,E1 -15950.951,E2 -15950.951} C_VEL
LIN {X 0,Y 317.312,Z 339.249,A -85,B 0,C 180,E1 -15952.634,E2 -15952.634} C_VEL
LIN {X 0,Y 318.204,Z 331.407,A -85,B 0,C 180,E1 -15953.827,E2 -15953.827} C_VEL
LIN {X 0,Y 318.174,Z 321.969,A -85,B 0,C 180,E1 -15955.27,E2 -15955.27} C_VEL
LIN {X 0,Y 317.191,Z 312.561,A -85,B 0,C 180,E1 -15956.743,E2 -15956.743} C_VEL
LIN {X 0,Y 315.072,Z 301.888,A -85,B 0,C 180,E1 -15958.508,E2 -15958.508} C_VEL
LIN {X 0,Y 313.034,Z 294.608,A -85,B 0,C 180,E1 -15959.829,E2 -15959.829} C_VEL
LIN {X 0,Y 311.888,Z 290.566,A -85,B 0,C 180,E1 -15960.578,E2 -15960.578} C_VEL
LIN {X 0,Y 310.484,Z 286.74,A -85,B 0,C 180,E1 -15961.374,E2 -15961.374} C_VEL
LIN {X 0,Y 310.223,Z 285.392,A -85,B 0,C 180,E1 -15961.604,E2 -15961.604} C_VEL
LIN {X 0,Y 308.471,Z 281.537,A -85,B 0,C 180,E1 -15962.543,E2 -15962.543} C_VEL
LIN {X 0,Y 308.014,Z 279.274,A -85,B 0,C 180,E1 -15962.948,E2 -15962.948} C_VEL
LIN {X 0,Y 308.666,Z 276.956,A -85,B 0,C 180,E1 -15964.947,E2 -15964.947} C_VEL
LIN {X 0,Y 309.173,Z 274.01,A -85,B 0,C 180,E1 -15967.862,E2 -15967.862} C_VEL
LIN {X 0,Y 309.228,Z 272.575,A -85,B 0,C 180,E1 -15969.522,E2 -15969.522} C_VEL
LIN {X 0,Y 309.132,Z 271.165,A -85,B 0,C 180,E1 -15971.389,E2 -15971.389} C_VEL
LIN {X 0,Y 308.78,Z 268.926,A -85,B 0,C 180,E1 -15975.124,E2 -15975.124} C_VEL
LIN {X 0,Y 308.428,Z 267.478,A -85,B 0,C 180,E1 -15978.638,E2 -15978.638} C_VEL
LIN {X 0,Y 308.158,Z 266.641,A -85,B 0,C 180,E1 -15981.992,E2 -15981.992} C_VEL
LIN {X 0,Y 307.892,Z 266.331,A -85,B 0,C 180,E1 -15985.26,E2 -15985.26} C_VEL
LIN {X 0,Y 307.472,Z 266.533,A -85,B 0,C 180,E1 -15988.053,E2 -15988.053} C_VEL
LIN {X 0,Y 308.612,Z 269.334,A -85,B 0,C 180,E1 -15988.824,E2 -15988.824} C_VEL
LIN {X 0,Y 310.655,Z 271.996,A -85,B 0,C 180,E1 -15989.845,E2 -15989.845} C_VEL
LIN {X 0,Y 311.908,Z 274.324,A -85,B 0,C 180,E1 -15990.53,E2 -15990.53} C_VEL
LIN {X 0,Y 313.082,Z 276.138,A -85,B 0,C 180,E1 -15991.101,E2 -15991.101} C_VEL
LIN {X 0,Y 317.074,Z 284.282,A -85,B 0,C 180,E1 -15993.213,E2 -15993.213} C_VEL
LIN {X 0,Y 319.588,Z 290.737,A -85,B 0,C 180,E1 -15994.675,E2 -15994.675} C_VEL
LIN {X 0,Y 321.775,Z 297.864,A -85,B 0,C 180,E1 -15996.183,E2 -15996.183} C_VEL
LIN {X 0,Y 322.869,Z 303.302,A -85,B 0,C 180,E1 -15997.254,E2 -15997.254} C_VEL
LIN {X 0,Y 322.823,Z 305.236,A -85,B 0,C 180,E1 -15997.57,E2 -15997.57} C_VEL
LIN {X 0,Y 319.98,Z 316.004,A -85,B 0,C 180,E1 -15999.089,E2 -15999.089} C_VEL
LIN {X 0,Y 317.386,Z 324.838,A -85,B 0,C 180,E1 -16000.601,E2 -16000.601} C_VEL
LIN {X 0,Y 314.702,Z 333.606,A -85,B 0,C 180,E1 -16002.453,E2 -16002.453} C_VEL
LIN {X 0,Y 311.954,Z 341.947,A -85,B 0,C 180,E1 -16004.65,E2 -16004.65} C_VEL
LIN {X 0,Y 309.627,Z 348.515,A -85,B 0,C 180,E1 -16006.881,E2 -16006.881} C_VEL
LIN {X 0,Y 307.567,Z 354.214,A -85,B 0,C 180,E1 -16009.467,E2 -16009.467} C_VEL
LIN {X 0,Y 306.577,Z 356.39,A -85,B 0,C 180,E1 -16010.766,E2 -16010.766} C_VEL
LIN {X 0,Y 305.57,Z 359.456,A -85,B 0,C 180,E1 -16013.397,E2 -16013.397} C_VEL
LIN {X 0,Y 305.112,Z 360.416,A -85,B 0,C 180,E1 -16014.714,E2 -16014.714} C_VEL
LIN {X 0,Y 304.803,Z 360.95,A -85,B 0,C 180,E1 -16016.034,E2 -16016.034} C_VEL
LIN {X 0,Y 304.099,Z 360.899,A -85,B 0,C 180,E1 -16018.676,E2 -16018.676} C_VEL
LIN {X 0,Y 303.945,Z 360.277,A -85,B 0,C 180,E1 -16020,E2 -16020} C_VEL
LIN {X 0,Y 303.859,Z 357.754,A -85,B 0,C 180,E1 -16022.652,E2 -16022.652} C_VEL
LIN {X 0,Y 303.956,Z 354.763,A -85,B 0,C 180,E1 -16024.642,E2 -16024.642} C_VEL
LIN {X 0,Y 304.107,Z 350.731,A -85,B 0,C 180,E1 -16026.636,E2 -16026.636} C_VEL
LIN {X 0,Y 304.471,Z 344.593,A -85,B 0,C 180,E1 -16028.964,E2 -16028.964} C_VEL
LIN {X 0,Y 304.975,Z 337.874,A -85,B 0,C 180,E1 -16030.96,E2 -16030.96} C_VEL
LIN {X 0,Y 305.707,Z 329.605,A -85,B 0,C 180,E1 -16032.953,E2 -16032.953} C_VEL
LIN {X 0,Y 306.479,Z 321.25,A -85,B 0,C 180,E1 -16034.611,E2 -16034.611} C_VEL
LIN {X 0,Y 307.333,Z 311.165,A -85,B 0,C 180,E1 -16036.267,E2 -16036.267} C_VEL
LIN {X 0,Y 308.354,Z 300.083,A -85,B 0,C 180,E1 -16037.749,E2 -16037.749} C_VEL
LIN {X 0,Y 309.41,Z 287.987,A -85,B 0,C 180,E1 -16039.058,E2 -16039.058} C_VEL
LIN {X 0,Y 309.246,Z 283.34,A -85,B 0,C 180,E1 -16039.499,E2 -16039.499} C_VEL
LIN {X 0,Y 306.719,Z 269.959,A -85,B 0,C 180,E1 -16040.629,E2 -16040.629} C_VEL
LIN {X 0,Y 304.242,Z 256.338,A -85,B 0,C 180,E1 -16041.512,E2 -16041.512} C_VEL
LIN {X 0,Y 304.137,Z 255.5,A -85,B 0,C 180,E1 -16041.575,E2 -16041.575} C_VEL
LIN {X 0,Y 304.258,Z 251.39,A -85,B 0,C 180,E1 -16046.033,E2 -16046.033} C_VEL
LIN {X 0,Y 304.341,Z 250.58,A -85,B 0,C 180,E1 -16047.507,E2 -16047.507} C_VEL
LIN {X 0,Y 304.85,Z 250.509,A -85,B 0,C 180,E1 -16052.022,E2 -16052.022} C_VEL
LIN {X 0,Y 305.248,Z 250.462,A -85,B 0,C 180,E1 -16055.142,E2 -16055.142} C_VEL
LIN {X 0,Y 305.431,Z 250.437,A -85,B 0,C 180,E1 -16058.524,E2 -16058.524} C_VEL
LIN {X 0,Y 305.444,Z 250.435,A -85,B 0,C 180,E1 -16061.857,E2 -16061.857} C_VEL
LIN {X 0,Y 305.403,Z 250.441,A -85,B 0,C 180,E1 -16065.511,E2 -16065.511} C_VEL
LIN {X 0,Y 305.415,Z 250.438,A -85,B 0,C 180,E1 -16068.138,E2 -16068.138} C_VEL
LIN {X 0,Y 305.462,Z 250.433,A -85,B 0,C 180,E1 -16071.595,E2 -16071.595} C_VEL
LIN {X 0,Y 305.464,Z 250.437,A -85,B 0,C 180,E1 -16074.887,E2 -16074.887} C_VEL
LIN {X 0,Y 305.445,Z 250.437,A -85,B 0,C 180,E1 -16078.358,E2 -16078.358} C_VEL
LIN {X 0,Y 305.494,Z 250.43,A -85,B 0,C 180,E1 -16081.111,E2 -16081.111} C_VEL
LIN {X 0,Y 305.511,Z 250.428,A -85,B 0,C 180,E1 -16084.082,E2 -16084.082} C_VEL
LIN {X 0,Y 305.485,Z 250.435,A -85,B 0,C 180,E1 -16088.401,E2 -16088.401} C_VEL
LIN {X 0,Y 305.593,Z 250.416,A -85,B 0,C 180,E1 -16091.218,E2 -16091.218} C_VEL
LIN {X 0,Y 305.652,Z 250.409,A -85,B 0,C 180,E1 -16095.349,E2 -16095.349} C_VEL
LIN {X 0,Y 305.627,Z 250.413,A -85,B 0,C 180,E1 -16099.399,E2 -16099.399} C_VEL
LIN {X 0,Y 305.749,Z 250.402,A -85,B 0,C 180,E1 -16102.072,E2 -16102.072} C_VEL
LIN {X 0,Y 305.657,Z 250.409,A -85,B 0,C 180,E1 -16104.723,E2 -16104.723} C_VEL
LIN {X 0,Y 305.946,Z 250.373,A -85,B 0,C 180,E1 -16108.684,E2 -16108.684} C_VEL
LIN {X 0,Y 305.938,Z 250.377,A -85,B 0,C 180,E1 -16111.316,E2 -16111.316} C_VEL
LIN {X 0,Y 305.627,Z 250.598,A -85,B 0,C 180,E1 -16113.79,E2 -16113.79} C_VEL
LIN {X 0,Y 305.866,Z 254.387,A -85,B 0,C 180,E1 -16115.935,E2 -16115.935} C_VEL
LIN {X 0,Y 305.454,Z 262.809,A -85,B 0,C 180,E1 -16120.607,E2 -16120.607} C_VEL
LIN {X 0,Y 305.174,Z 270.158,A -85,B 0,C 180,E1 -16124.705,E2 -16124.705} C_VEL
LIN {X 0,Y 304.935,Z 277.554,A -85,B 0,C 180,E1 -16128.824,E2 -16128.824} C_VEL
LIN {X 0,Y 304.883,Z 278.554,A -85,B 0,C 180,E1 -16129.357,E2 -16129.357} C_VEL
LIN {X 0,Y 306.725,Z 288.352,A -85,B 0,C 180,E1 -16129.923,E2 -16129.923} C_VEL
LIN {X 0,Y 308.334,Z 297.987,A -85,B 0,C 180,E1 -16130.663,E2 -16130.663} C_VEL
LIN {X 0,Y 309.014,Z 303.496,A -85,B 0,C 180,E1 -16131.175,E2 -16131.175} C_VEL
LIN {X 0,Y 308.416,Z 312.362,A -85,B 0,C 180,E1 -16132.086,E2 -16132.086} C_VEL
LIN {X 0,Y 307.687,Z 320.698,A -85,B 0,C 180,E1 -16133.152,E2 -16133.152} C_VEL
LIN {X 0,Y 306.795,Z 330.344,A -85,B 0,C 180,E1 -16134.713,E2 -16134.713} C_VEL
LIN {X 0,Y 305.944,Z 338.26,A -85,B 0,C 180,E1 -16136.376,E2 -16136.376} C_VEL
LIN {X 0,Y 305.318,Z 343.613,A -85,B 0,C 180,E1 -16137.763,E2 -16137.763} C_VEL
LIN {X 0,Y 304.815,Z 348.54,A -85,B 0,C 180,E1 -16139.337,E2 -16139.337} C_VEL
LIN {X 0,Y 304.312,Z 353.312,A -85,B 0,C 180,E1 -16141.294,E2 -16141.294} C_VEL
LIN {X 0,Y 304.021,Z 356.104,A -85,B 0,C 180,E1 -16142.866,E2 -16142.866} C_VEL
LIN {X 0,Y 303.703,Z 358.854,A -85,B 0,C 180,E1 -16145.347,E2 -16145.347} C_VEL
LIN {X 0,Y 303.631,Z 359.728,A -85,B 0,C 180,E1 -16147,E2 -16147} C_VEL
LIN {X 0,Y 303.725,Z 359.816,A -85,B 0,C 180,E1 -16148.665,E2 -16148.665} C_VEL
LIN {X 0,Y 303.964,Z 359.101,A -85,B 0,C 180,E1 -16150.345,E2 -16150.345} C_VEL
LIN {X 0,Y 304.421,Z 357.164,A -85,B 0,C 180,E1 -16152.373,E2 -16152.373} C_VEL
LIN {X 0,Y 305.027,Z 353.958,A -85,B 0,C 180,E1 -16154.417,E2 -16154.417} C_VEL
LIN {X 0,Y 305.817,Z 349.3,A -85,B 0,C 180,E1 -16156.414,E2 -16156.414} C_VEL
LIN {X 0,Y 306.537,Z 345.113,A -85,B 0,C 180,E1 -16157.818,E2 -16157.818} C_VEL
LIN {X 0,Y 307.497,Z 338.997,A -85,B 0,C 180,E1 -16159.459,E2 -16159.459} C_VEL
LIN {X 0,Y 308.844,Z 330.757,A -85,B 0,C 180,E1 -16161.205,E2 -16161.205} C_VEL
LIN {X 0,Y 309.954,Z 322.715,A -85,B 0,C 180,E1 -16162.523,E2 -16162.523} C_VEL
LIN {X 0,Y 310.938,Z 314.3,A -85,B 0,C 180,E1 -16163.631,E2 -16163.631} C_VEL
LIN {X 0,Y 311.558,Z 306.784,A -85,B 0,C 180,E1 -16164.449,E2 -16164.449} C_VEL
LIN {X 0,Y 310.364,Z 298.698,A -85,B 0,C 180,E1 -16165.299,E2 -16165.299} C_VEL
LIN {X 0,Y 308.431,Z 289.642,A -85,B 0,C 180,E1 -16166.111,E2 -16166.111} C_VEL
LIN {X 0,Y 305.701,Z 279.801,A -85,B 0,C 180,E1 -16166.857,E2 -16166.857} C_VEL
LIN {X 0,Y 306.091,Z 272.156,A -85,B 0,C 180,E1 -16171.172,E2 -16171.172} C_VEL
LIN {X 0,Y 306.292,Z 266.892,A -85,B 0,C 180,E1 -16174.153,E2 -16174.153} C_VEL
LIN {X 0,Y 306.604,Z 261.636,A -85,B 0,C 180,E1 -16177.065,E2 -16177.065} C_VEL
LIN {X 0,Y 306.732,Z 259.176,A -85,B 0,C 180,E1 -16178.409,E2 -16178.409} C_VEL
LIN {X 0,Y 306.088,Z 257.498,A -85,B 0,C 180,E1 -16179.457,E2 -16179.457} C_VEL
LIN {X 0,Y 304.391,Z 256.171,A -85,B 0,C 180,E1 -16180.496,E2 -16180.496} C_VEL
LIN {X 0,Y 300.187,Z 253.845,A -85,B 0,C 180,E1 -16182.59,E2 -16182.59} C_VEL
LIN {X 0,Y 298.834,Z 252.379,A -85,B 0,C 180,E1 -16183.674,E2 -16183.674} C_VEL
LIN {X 0,Y 298.645,Z 251.798,A -85,B 0,C 180,E1 -16184.04,E2 -16184.04} C_VEL
LIN {X 0,Y 298.589,Z 251.293,A -85,B 0,C 180,E1 -16184.365,E2 -16184.365} C_VEL
LIN {X 0,Y 298.557,Z 251.299,A -85,B 0,C 180,E1 -16187.768,E2 -16187.768} C_VEL
LIN {X 0,Y 298.734,Z 251.277,A -85,B 0,C 180,E1 -16191.885,E2 -16191.885} C_VEL
LIN {X 0,Y 298.644,Z 251.286,A -85,B 0,C 180,E1 -16194.598,E2 -16194.598} C_VEL
LIN {X 0,Y 298.924,Z 251.252,A -85,B 0,C 180,E1 -16198.653,E2 -16198.653} C_VEL
LIN {X 0,Y 298.924,Z 251.249,A -85,B 0,C 180,E1 -16201.347,E2 -16201.347} C_VEL
LIN {X 0,Y 298.645,Z 251.285,A -85,B 0,C 180,E1 -16205.401,E2 -16205.401} C_VEL
LIN {X 0,Y 298.714,Z 251.275,A -85,B 0,C 180,E1 -16208.115,E2 -16208.115} C_VEL
LIN {X 0,Y 298.556,Z 251.297,A -85,B 0,C 180,E1 -16212.231,E2 -16212.231} C_VEL
LIN {X 0,Y 298.607,Z 251.29,A -85,B 0,C 180,E1 -16215.209,E2 -16215.209} C_VEL
LIN {X 0,Y 298.54,Z 251.296,A -85,B 0,C 180,E1 -16219.243,E2 -16219.243} C_VEL
LIN {X 0,Y 298.43,Z 251.311,A -85,B 0,C 180,E1 -16223.6,E2 -16223.6} C_VEL
LIN {X 0,Y 298.49,Z 251.301,A -85,B 0,C 180,E1 -16226.574,E2 -16226.574} C_VEL
LIN {X 0,Y 298.422,Z 251.309,A -85,B 0,C 180,E1 -16229.641,E2 -16229.641} C_VEL
LIN {X 0,Y 298.397,Z 251.315,A -85,B 0,C 180,E1 -16232.8,E2 -16232.8} C_VEL
LIN {X 0,Y 298.447,Z 251.307,A -85,B 0,C 180,E1 -16236.808,E2 -16236.808} C_VEL
LIN {X 0,Y 298.409,Z 251.311,A -85,B 0,C 180,E1 -16239.486,E2 -16239.486} C_VEL
LIN {X 0,Y 298.444,Z 251.309,A -85,B 0,C 180,E1 -16244.002,E2 -16244.002} C_VEL
LIN {X 0,Y 298.497,Z 251.471,A -85,B 0,C 180,E1 -16244.7,E2 -16244.7} C_VEL
LIN {X 0,Y 299.541,Z 257.284,A -85,B 0,C 180,E1 -16248.932,E2 -16248.932} C_VEL
LIN {X 0,Y 300.208,Z 261.195,A -85,B 0,C 180,E1 -16251.656,E2 -16251.656} C_VEL
LIN {X 0,Y 300.388,Z 264.992,A -85,B 0,C 180,E1 -16254.203,E2 -16254.203} C_VEL
LIN {X 0,Y 299.573,Z 270.316,A -85,B 0,C 180,E1 -16257.625,E2 -16257.625} C_VEL
LIN {X 0,Y 298.712,Z 275.953,A -85,B 0,C 180,E1 -16261.186,E2 -16261.186} C_VEL
LIN {X 0,Y 297.988,Z 281.863,A -85,B 0,C 180,E1 -16264.879,E2 -16264.879} C_VEL
LIN {X 0,Y 297.605,Z 285.618,A -85,B 0,C 180,E1 -16267.153,E2 -16267.153} C_VEL
LIN {X 0,Y 298.546,Z 296.381,A -85,B 0,C 180,E1 -16268.962,E2 -16268.962} C_VEL
LIN {X 0,Y 298.509,Z 300.516,A -85,B 0,C 180,E1 -16269.54,E2 -16269.54} C_VEL
LIN {X 0,Y 300.442,Z 315.731,A -85,B 0,C 180,E1 -16270.29,E2 -16270.29} C_VEL
LIN {X 0,Y 301.595,Z 326.035,A -85,B 0,C 180,E1 -16271.048,E2 -16271.048} C_VEL
LIN {X 0,Y 302.036,Z 331.516,A -85,B 0,C 180,E1 -16271.516,E2 -16271.516} C_VEL
LIN {X 0,Y 301.254,Z 341.749,A -85,B 0,C 180,E1 -16272.521,E2 -16272.521} C_VEL
LIN {X 0,Y 300.348,Z 350.541,A -85,B 0,C 180,E1 -16273.614,E2 -16273.614} C_VEL
LIN {X 0,Y 299.767,Z 356.452,A -85,B 0,C 180,E1 -16274.504,E2 -16274.504} C_VEL
LIN {X 0,Y 299.042,Z 363.224,A -85,B 0,C 180,E1 -16275.714,E2 -16275.714} C_VEL
LIN {X 0,Y 298.349,Z 369.516,A -85,B 0,C 180,E1 -16277.069,E2 -16277.069} C_VEL
LIN {X 0,Y 297.711,Z 374.775,A -85,B 0,C 180,E1 -16278.425,E2 -16278.425} C_VEL
LIN {X 0,Y 297.334,Z 379.175,A -85,B 0,C 180,E1 -16279.789,E2 -16279.789} C_VEL
LIN {X 0,Y 296.911,Z 384.392,A -85,B 0,C 180,E1 -16281.835,E2 -16281.835} C_VEL
LIN {X 0,Y 296.761,Z 387.044,A -85,B 0,C 180,E1 -16283.2,E2 -16283.2} C_VEL
LIN {X 0,Y 296.7,Z 389.134,A -85,B 0,C 180,E1 -16284.563,E2 -16284.563} C_VEL
LIN {X 0,Y 296.696,Z 390.7,A -85,B 0,C 180,E1 -16285.925,E2 -16285.925} C_VEL
LIN {X 0,Y 296.748,Z 391.726,A -85,B 0,C 180,E1 -16287.285,E2 -16287.285} C_VEL
LIN {X 0,Y 296.83,Z 392.159,A -85,B 0,C 180,E1 -16288.643,E2 -16288.643} C_VEL
LIN {X 0,Y 296.97,Z 392.086,A -85,B 0,C 180,E1 -16290,E2 -16290} C_VEL
LIN {X 0,Y 296.635,Z 392.855,A -85,B 0,C 180,E1 -16292.716,E2 -16292.716} C_VEL
LIN {X 0,Y 296.608,Z 392.715,A -85,B 0,C 180,E1 -16294.076,E2 -16294.076} C_VEL
LIN {X 0,Y 296.655,Z 391.254,A -85,B 0,C 180,E1 -16296.803,E2 -16296.803} C_VEL
LIN {X 0,Y 296.877,Z 389.932,A -85,B 0,C 180,E1 -16298.166,E2 -16298.166} C_VEL
LIN {X 0,Y 297.68,Z 386.036,A -85,B 0,C 180,E1 -16300.887,E2 -16300.887} C_VEL
LIN {X 0,Y 298.657,Z 382.028,A -85,B 0,C 180,E1 -16302.918,E2 -16302.918} C_VEL
LIN {X 0,Y 300.29,Z 377.001,A -85,B 0,C 180,E1 -16304.919,E2 -16304.919} C_VEL
LIN {X 0,Y 302.231,Z 369.817,A -85,B 0,C 180,E1 -16307.238,E2 -16307.238} C_VEL
LIN {X 0,Y 305.018,Z 360.819,A -85,B 0,C 180,E1 -16309.518,E2 -16309.518} C_VEL
LIN {X 0,Y 308.01,Z 351.475,A -85,B 0,C 180,E1 -16311.413,E2 -16311.413} C_VEL
LIN {X 0,Y 311.205,Z 340.295,A -85,B 0,C 180,E1 -16313.279,E2 -16313.279} C_VEL
LIN {X 0,Y 312.148,Z 333.248,A -85,B 0,C 180,E1 -16314.419,E2 -16314.419} C_VEL
LIN {X 0,Y 312.326,Z 323.383,A -85,B 0,C 180,E1 -16316.026,E2 -16316.026} C_VEL
LIN {X 0,Y 311.25,Z 312.496,A -85,B 0,C 180,E1 -16317.871,E2 -16317.871} C_VEL
LIN {X 0,Y 309.265,Z 302.535,A -85,B 0,C 180,E1 -16319.698,E2 -16319.698} C_VEL
LIN {X 0,Y 307.479,Z 295.298,A -85,B 0,C 180,E1 -16321.122,E2 -16321.122} C_VEL
LIN {X 0,Y 305.566,Z 289.324,A -85,B 0,C 180,E1 -16322.461,E2 -16322.461} C_VEL
LIN {X 0,Y 303.812,Z 284.079,A -85,B 0,C 180,E1 -16323.724,E2 -16323.724} C_VEL
LIN {X 0,Y 302.583,Z 281.497,A -85,B 0,C 180,E1 -16324.512,E2 -16324.512} C_VEL
LIN {X 0,Y 301.788,Z 277.992,A -85,B 0,C 180,E1 -16325.337,E2 -16325.337} C_VEL
LIN {X 0,Y 302.235,Z 275.613,A -85,B 0,C 180,E1 -16327.757,E2 -16327.757} C_VEL
LIN {X 0,Y 302.241,Z 273.28,A -85,B 0,C 180,E1 -16330.624,E2 -16330.624} C_VEL
LIN {X 0,Y 301.904,Z 270.961,A -85,B 0,C 180,E1 -16334.297,E2 -16334.297} C_VEL
LIN {X 0,Y 301.626,Z 269.497,A -85,B 0,C 180,E1 -16337.491,E2 -16337.491} C_VEL
LIN {X 0,Y 301.336,Z 268.448,A -85,B 0,C 180,E1 -16340.971,E2 -16340.971} C_VEL
LIN {X 0,Y 301.052,Z 267.951,A -85,B 0,C 180,E1 -16344.294,E2 -16344.294} C_VEL
LIN {X 0,Y 300.928,Z 267.943,A -85,B 0,C 180,E1 -16345.493,E2 -16345.493} C_VEL
LIN {X 0,Y 301.363,Z 269.416,A -85,B 0,C 180,E1 -16345.965,E2 -16345.965} C_VEL
LIN {X 0,Y 304.396,Z 273.517,A -85,B 0,C 180,E1 -16347.925,E2 -16347.925} C_VEL
LIN {X 0,Y 305.137,Z 275.163,A -85,B 0,C 180,E1 -16348.452,E2 -16348.452} C_VEL
LIN {X 0,Y 306.815,Z 277.457,A -85,B 0,C 180,E1 -16349.397,E2 -16349.397} C_VEL
LIN {X 0,Y 310.866,Z 285.543,A -85,B 0,C 180,E1 -16351.85,E2 -16351.85} C_VEL
LIN {X 0,Y 313.7,Z 292.575,A -85,B 0,C 180,E1 -16353.657,E2 -16353.657} C_VEL
LIN {X 0,Y 316.258,Z 301.302,A -85,B 0,C 180,E1 -16355.661,E2 -16355.661} C_VEL
LIN {X 0,Y 317.098,Z 307.116,A -85,B 0,C 180,E1 -16356.866,E2 -16356.866} C_VEL
LIN {X 0,Y 314.304,Z 317.161,A -85,B 0,C 180,E1 -16358.349,E2 -16358.349} C_VEL
LIN {X 0,Y 311.015,Z 327.381,A -85,B 0,C 180,E1 -16360.187,E2 -16360.187} C_VEL
LIN {X 0,Y 308.215,Z 335.747,A -85,B 0,C 180,E1 -16362.072,E2 -16362.072} C_VEL
LIN {X 0,Y 305.719,Z 342.691,A -85,B 0,C 180,E1 -16363.987,E2 -16363.987} C_VEL
LIN {X 0,Y 303.544,Z 348.36,A -85,B 0,C 180,E1 -16365.93,E2 -16365.93} C_VEL
LIN {X 0,Y 301.393,Z 353.761,A -85,B 0,C 180,E1 -16368.345,E2 -16368.345} C_VEL
LIN {X 0,Y 299.657,Z 357.424,A -85,B 0,C 180,E1 -16370.551,E2 -16370.551} C_VEL
LIN {X 0,Y 299.102,Z 359.043,A -85,B 0,C 180,E1 -16371.895,E2 -16371.895} C_VEL
LIN {X 0,Y 298.58,Z 360.261,A -85,B 0,C 180,E1 -16373.241,E2 -16373.241} C_VEL
LIN {X 0,Y 297.762,Z 361.523,A -85,B 0,C 180,E1 -16375.94,E2 -16375.94} C_VEL
LIN {X 0,Y 297.329,Z 361.604,A -85,B 0,C 180,E1 -16377.291,E2 -16377.291} C_VEL
LIN {X 0,Y 297.011,Z 361.275,A -85,B 0,C 180,E1 -16378.644,E2 -16378.644} C_VEL
LIN {X 0,Y 296.764,Z 359.368,A -85,B 0,C 180,E1 -16381.357,E2 -16381.357} C_VEL
LIN {X 0,Y 296.778,Z 357.825,A -85,B 0,C 180,E1 -16382.715,E2 -16382.715} C_VEL
LIN {X 0,Y 296.877,Z 354.67,A -85,B 0,C 180,E1 -16384.753,E2 -16384.753} C_VEL
LIN {X 0,Y 297.11,Z 349.333,A -85,B 0,C 180,E1 -16387.257,E2 -16387.257} C_VEL
LIN {X 0,Y 297.521,Z 343.028,A -85,B 0,C 180,E1 -16389.518,E2 -16389.518} C_VEL
LIN {X 0,Y 298.053,Z 335.883,A -85,B 0,C 180,E1 -16391.562,E2 -16391.562} C_VEL
LIN {X 0,Y 298.901,Z 327.03,A -85,B 0,C 180,E1 -16393.599,E2 -16393.599} C_VEL
LIN {X 0,Y 299.84,Z 316.6,A -85,B 0,C 180,E1 -16395.555,E2 -16395.555} C_VEL
LIN {X 0,Y 300.758,Z 306.016,A -85,B 0,C 180,E1 -16397.159,E2 -16397.159} C_VEL
LIN {X 0,Y 301.818,Z 293.719,A -85,B 0,C 180,E1 -16398.674,E2 -16398.674} C_VEL
LIN {X 0,Y 302.45,Z 285.597,A -85,B 0,C 180,E1 -16399.49,E2 -16399.49} C_VEL
LIN {X 0,Y 300.293,Z 273.612,A -85,B 0,C 180,E1 -16400.583,E2 -16400.583} C_VEL
LIN {X 0,Y 297.578,Z 258.925,A -85,B 0,C 180,E1 -16401.613,E2 -16401.613} C_VEL
LIN {X 0,Y 297.055,Z 255.891,A -85,B 0,C 180,E1 -16401.786,E2 -16401.786} C_VEL
LIN {X 0,Y 297.197,Z 251.469,A -85,B 0,C 180,E1 -16406.699,E2 -16406.699} C_VEL
LIN {X 0,Y 297.519,Z 251.425,A -85,B 0,C 180,E1 -16409.74,E2 -16409.74} C_VEL
LIN {X 0,Y 297.913,Z 251.374,A -85,B 0,C 180,E1 -16412.86,E2 -16412.86} C_VEL
LIN {X 0,Y 298.288,Z 251.326,A -85,B 0,C 180,E1 -16416.088,E2 -16416.088} C_VEL
LIN {X 0,Y 298.4,Z 251.315,A -85,B 0,C 180,E1 -16419.488,E2 -16419.488} C_VEL
LIN {X 0,Y 298.402,Z 251.317,A -85,B 0,C 180,E1 -16423.103,E2 -16423.103} C_VEL
LIN {X 0,Y 298.374,Z 251.32,A -85,B 0,C 180,E1 -16426.915,E2 -16426.915} C_VEL
LIN {X 0,Y 298.387,Z 251.318,A -85,B 0,C 180,E1 -16431.011,E2 -16431.011} C_VEL
LIN {X 0,Y 298.407,Z 251.311,A -85,B 0,C 180,E1 -16433.928,E2 -16433.928} C_VEL
LIN {X 0,Y 298.396,Z 251.314,A -85,B 0,C 180,E1 -16437.199,E2 -16437.199} C_VEL
LIN {X 0,Y 298.414,Z 251.316,A -85,B 0,C 180,E1 -16440.622,E2 -16440.622} C_VEL
LIN {X 0,Y 298.453,Z 251.307,A -85,B 0,C 180,E1 -16444.921,E2 -16444.921} C_VEL
LIN {X 0,Y 298.443,Z 251.307,A -85,B 0,C 180,E1 -16449.314,E2 -16449.314} C_VEL
LIN {X 0,Y 298.541,Z 251.298,A -85,B 0,C 180,E1 -16452.179,E2 -16452.179} C_VEL
LIN {X 0,Y 298.597,Z 251.288,A -85,B 0,C 180,E1 -16454.995,E2 -16454.995} C_VEL
LIN {X 0,Y 298.586,Z 251.29,A -85,B 0,C 180,E1 -16459.146,E2 -16459.146} C_VEL
LIN {X 0,Y 298.7,Z 251.28,A -85,B 0,C 180,E1 -16461.884,E2 -16461.884} C_VEL
LIN {X 0,Y 298.627,Z 251.285,A -85,B 0,C 180,E1 -16464.598,E2 -16464.598} C_VEL
LIN {X 0,Y 298.912,Z 251.25,A -85,B 0,C 180,E1 -16468.653,E2 -16468.653} C_VEL
LIN {X 0,Y 298.905,Z 251.253,A -85,B 0,C 180,E1 -16471.347,E2 -16471.347} C_VEL
LIN {X 0,Y 298.635,Z 251.415,A -85,B 0,C 180,E1 -16473.542,E2 -16473.542} C_VEL
LIN {X 0,Y 298.85,Z 255.855,A -85,B 0,C 180,E1 -16476.075,E2 -16476.075} C_VEL
LIN {X 0,Y 298.469,Z 263.111,A -85,B 0,C 180,E1 -16480.172,E2 -16480.172} C_VEL
LIN {X 0,Y 298.176,Z 270.355,A -85,B 0,C 180,E1 -16484.252,E2 -16484.252} C_VEL
LIN {X 0,Y 297.961,Z 276.756,A -85,B 0,C 180,E1 -16487.856,E2 -16487.856} C_VEL
LIN {X 0,Y 297.89,Z 279.013,A -85,B 0,C 180,E1 -16489.026,E2 -16489.026} C_VEL
LIN {X 0,Y 299.726,Z 288.806,A -85,B 0,C 180,E1 -16489.609,E2 -16489.609} C_VEL
LIN {X 0,Y 301.224,Z 297.707,A -85,B 0,C 180,E1 -16490.307,E2 -16490.307} C_VEL
LIN {X 0,Y 302.068,Z 304.44,A -85,B 0,C 180,E1 -16490.946,E2 -16490.946} C_VEL
LIN {X 0,Y 301.53,Z 311.987,A -85,B 0,C 180,E1 -16491.735,E2 -16491.735} C_VEL
LIN {X 0,Y 300.904,Z 319.328,A -85,B 0,C 180,E1 -16492.667,E2 -16492.667} C_VEL
LIN {X 0,Y 300.223,Z 326.201,A -85,B 0,C 180,E1 -16493.717,E2 -16493.717} C_VEL
LIN {X 0,Y 299.543,Z 333.065,A -85,B 0,C 180,E1 -16494.981,E2 -16494.981} C_VEL
LIN {X 0,Y 298.725,Z 340.324,A -85,B 0,C 180,E1 -16496.617,E2 -16496.617} C_VEL
LIN {X 0,Y 297.931,Z 347.253,A -85,B 0,C 180,E1 -16498.647,E2 -16498.647} C_VEL
LIN {X 0,Y 297.609,Z 350.276,A -85,B 0,C 180,E1 -16499.73,E2 -16499.73} C_VEL
LIN {X 0,Y 297.14,Z 354.403,A -85,B 0,C 180,E1 -16501.626,E2 -16501.626} C_VEL
LIN {X 0,Y 296.901,Z 356.688,A -85,B 0,C 180,E1 -16502.986,E2 -16502.986} C_VEL
LIN {X 0,Y 296.67,Z 358.682,A -85,B 0,C 180,E1 -16504.649,E2 -16504.649} C_VEL
LIN {X 0,Y 296.557,Z 359.899,A -85,B 0,C 180,E1 -16506.332,E2 -16506.332} C_VEL
LIN {X 0,Y 296.648,Z 360.249,A -85,B 0,C 180,E1 -16508.572,E2 -16508.572} C_VEL
LIN {X 0,Y 296.782,Z 359.984,A -85,B 0,C 180,E1 -16509.745,E2 -16509.745} C_VEL
LIN {X 0,Y 297.138,Z 358.806,A -85,B 0,C 180,E1 -16511.473,E2 -16511.473} C_VEL
LIN {X 0,Y 297.596,Z 356.737,A -85,B 0,C 180,E1 -16513.225,E2 -16513.225} C_VEL
LIN {X 0,Y 298.174,Z 353.674,A -85,B 0,C 180,E1 -16515,E2 -16515} C_VEL
LIN {X 0,Y 298.905,Z 349.492,A -85,B 0,C 180,E1 -16516.793,E2 -16516.793} C_VEL
LIN {X 0,Y 299.658,Z 345.465,A -85,B 0,C 180,E1 -16518.165,E2 -16518.165} C_VEL
LIN {X 0,Y 300.553,Z 340.084,A -85,B 0,C 180,E1 -16519.662,E2 -16519.662} C_VEL
LIN {X 0,Y 301.606,Z 334.127,A -85,B 0,C 180,E1 -16521.012,E2 -16521.012} C_VEL
LIN {X 0,Y 302.744,Z 326.889,A -85,B 0,C 180,E1 -16522.357,E2 -16522.357} C_VEL
LIN {X 0,Y 303.91,Z 318.144,A -85,B 0,C 180,E1 -16523.675,E2 -16523.675} C_VEL
LIN {X 0,Y 304.925,Z 308.37,A -85,B 0,C 180,E1 -16524.815,E2 -16524.815} C_VEL
LIN {X 0,Y 303.634,Z 299.57,A -85,B 0,C 180,E1 -16525.781,E2 -16525.781} C_VEL
LIN {X 0,Y 301.731,Z 290.692,A -85,B 0,C 180,E1 -16526.613,E2 -16526.613} C_VEL
LIN {X 0,Y 299.268,Z 282.07,A -85,B 0,C 180,E1 -16527.307,E2 -16527.307} C_VEL
LIN {X 0,Y 298.787,Z 280.1,A -85,B 0,C 180,E1 -16527.482,E2 -16527.482} C_VEL
LIN {X 0,Y 299.151,Z 273.605,A -85,B 0,C 180,E1 -16531.209,E2 -16531.209} C_VEL
LIN {X 0,Y 299.368,Z 268.299,A -85,B 0,C 180,E1 -16534.258,E2 -16534.258} C_VEL
LIN {X 0,Y 299.79,Z 261.689,A -85,B 0,C 180,E1 -16537.97,E2 -16537.97} C_VEL
LIN {X 0,Y 299.779,Z 258.762,A -85,B 0,C 180,E1 -16539.678,E2 -16539.678} C_VEL
LIN {X 0,Y 298.995,Z 253.655,A -85,B 0,C 180,E1 -16542.913,E2 -16542.913} C_VEL
LIN {X 0,Y 298.645,Z 251.798,A -85,B 0,C 180,E1 -16544.04,E2 -16544.04} C_VEL
LIN {X 0,Y 298.155,Z 251.345,A -85,B 0,C 180,E1 -16544.767,E2 -16544.767} C_VEL
LIN {X 0,Y 296.095,Z 251.604,A -85,B 0,C 180,E1 -16546.232,E2 -16546.232} C_VEL
LIN {X 0,Y 292.537,Z 252.145,A -85,B 0,C 180,E1 -16548.467,E2 -16548.467} C_VEL
LIN {X 0,Y 291.609,Z 252.173,A -85,B 0,C 180,E1 -16549.632,E2 -16549.632} C_VEL
LIN {X 0,Y 291.557,Z 252.17,A -85,B 0,C 180,E1 -16550.026,E2 -16550.026} C_VEL
LIN {X 0,Y 291.706,Z 252.151,A -85,B 0,C 180,E1 -16553.081,E2 -16553.081} C_VEL
LIN {X 0,Y 291.89,Z 252.128,A -85,B 0,C 180,E1 -16558.62,E2 -16558.62} C_VEL
LIN {X 0,Y 291.89,Z 252.125,A -85,B 0,C 180,E1 -16561.38,E2 -16561.38} C_VEL
LIN {X 0,Y 291.613,Z 252.161,A -85,B 0,C 180,E1 -16565.532,E2 -16565.532} C_VEL
LIN {X 0,Y 291.675,Z 252.152,A -85,B 0,C 180,E1 -16568.919,E2 -16568.919} C_VEL
LIN {X 0,Y 291.523,Z 252.173,A -85,B 0,C 180,E1 -16572.531,E2 -16572.531} C_VEL
LIN {X 0,Y 291.557,Z 252.167,A -85,B 0,C 180,E1 -16575.376,E2 -16575.376} C_VEL
LIN {X 0,Y 291.452,Z 252.181,A -85,B 0,C 180,E1 -16579.875,E2 -16579.875} C_VEL
LIN {X 0,Y 291.384,Z 252.186,A -85,B 0,C 180,E1 -16584.207,E2 -16584.207} C_VEL
LIN {X 0,Y 291.424,Z 252.181,A -85,B 0,C 180,E1 -16587.271,E2 -16587.271} C_VEL
LIN {X 0,Y 291.339,Z 252.195,A -85,B 0,C 180,E1 -16590.437,E2 -16590.437} C_VEL
LIN {X 0,Y 291.346,Z 252.193,A -85,B 0,C 180,E1 -16593.698,E2 -16593.698} C_VEL
LIN {X 0,Y 291.382,Z 252.186,A -85,B 0,C 180,E1 -16597.255,E2 -16597.255} C_VEL
LIN {X 0,Y 291.335,Z 252.196,A -85,B 0,C 180,E1 -16600.642,E2 -16600.642} C_VEL
LIN {X 0,Y 291.453,Z 252.386,A -85,B 0,C 180,E1 -16604.613,E2 -16604.613} C_VEL
LIN {X 0,Y 292.332,Z 257.14,A -85,B 0,C 180,E1 -16608.183,E2 -16608.183} C_VEL
LIN {X 0,Y 293.111,Z 261.652,A -85,B 0,C 180,E1 -16611.435,E2 -16611.435} C_VEL
LIN {X 0,Y 293.34,Z 265.317,A -85,B 0,C 180,E1 -16613.953,E2 -16613.953} C_VEL
LIN {X 0,Y 292.593,Z 270.244,A -85,B 0,C 180,E1 -16617.213,E2 -16617.213} C_VEL
LIN {X 0,Y 291.62,Z 276.349,A -85,B 0,C 180,E1 -16621.184,E2 -16621.184} C_VEL
LIN {X 0,Y 290.876,Z 282.263,A -85,B 0,C 180,E1 -16624.987,E2 -16624.987} C_VEL
LIN {X 0,Y 290.701,Z 284.172,A -85,B 0,C 180,E1 -16626.151,E2 -16626.151} C_VEL
LIN {X 0,Y 291.889,Z 296.965,A -85,B 0,C 180,E1 -16628.458,E2 -16628.458} C_VEL
LIN {X 0,Y 291.828,Z 300.134,A -85,B 0,C 180,E1 -16628.919,E2 -16628.919} C_VEL
LIN {X 0,Y 293.712,Z 315.023,A -85,B 0,C 180,E1 -16629.678,E2 -16629.678} C_VEL
LIN {X 0,Y 294.807,Z 325.914,A -85,B 0,C 180,E1 -16630.504,E2 -16630.504} C_VEL
LIN {X 0,Y 295.231,Z 333.993,A -85,B 0,C 180,E1 -16631.254,E2 -16631.254} C_VEL
LIN {X 0,Y 294.503,Z 342.196,A -85,B 0,C 180,E1 -16632.107,E2 -16632.107} C_VEL
LIN {X 0,Y 293.658,Z 350.173,A -85,B 0,C 180,E1 -16633.131,E2 -16633.131} C_VEL
LIN {X 0,Y 292.885,Z 356.981,A -85,B 0,C 180,E1 -16634.192,E2 -16634.192} C_VEL
LIN {X 0,Y 291.983,Z 365.003,A -85,B 0,C 180,E1 -16635.717,E2 -16635.717} C_VEL
LIN {X 0,Y 291.045,Z 372.319,A -85,B 0,C 180,E1 -16637.448,E2 -16637.448} C_VEL
LIN {X 0,Y 290.512,Z 377.051,A -85,B 0,C 180,E1 -16638.841,E2 -16638.841} C_VEL
LIN {X 0,Y 289.986,Z 382.641,A -85,B 0,C 180,E1 -16640.937,E2 -16640.937} C_VEL
LIN {X 0,Y 289.683,Z 386.797,A -85,B 0,C 180,E1 -16643.033,E2 -16643.033} C_VEL
LIN {X 0,Y 289.625,Z 388.844,A -85,B 0,C 180,E1 -16644.43,E2 -16644.43} C_VEL
LIN {X 0,Y 289.609,Z 390.369,A -85,B 0,C 180,E1 -16645.825,E2 -16645.825} C_VEL
LIN {X 0,Y 289.663,Z 391.379,A -85,B 0,C 180,E1 -16647.219,E2 -16647.219} C_VEL
LIN {X 0,Y 289.734,Z 391.792,A -85,B 0,C 180,E1 -16648.61,E2 -16648.61} C_VEL
LIN {X 0,Y 289.878,Z 391.688,A -85,B 0,C 180,E1 -16650,E2 -16650} C_VEL
LIN {X 0,Y 289.556,Z 392.339,A -85,B 0,C 180,E1 -16652.783,E2 -16652.783} C_VEL
LIN {X 0,Y 289.522,Z 392.304,A -85,B 0,C 180,E1 -16654.176,E2 -16654.176} C_VEL
LIN {X 0,Y 289.58,Z 390.996,A -85,B 0,C 180,E1 -16656.97,E2 -16656.97} C_VEL
LIN {X 0,Y 290.163,Z 388.161,A -85,B 0,C 180,E1 -16659.762,E2 -16659.762} C_VEL
LIN {X 0,Y 290.988,Z 384.957,A -85,B 0,C 180,E1 -16661.847,E2 -16661.847} C_VEL
LIN {X 0,Y 292.216,Z 380.813,A -85,B 0,C 180,E1 -16663.917,E2 -16663.917} C_VEL
LIN {X 0,Y 294.033,Z 375.65,A -85,B 0,C 180,E1 -16665.955,E2 -16665.955} C_VEL
LIN {X 0,Y 295.885,Z 369.442,A -85,B 0,C 180,E1 -16667.986,E2 -16667.986} C_VEL
LIN {X 0,Y 298.913,Z 360.594,A -85,B 0,C 180,E1 -16670.292,E2 -16670.292} C_VEL
LIN {X 0,Y 302.663,Z 349.714,A -85,B 0,C 180,E1 -16672.529,E2 -16672.529} C_VEL
LIN {X 0,Y 305.389,Z 340.48,A -85,B 0,C 180,E1 -16674.11,E2 -16674.11} C_VEL
LIN {X 0,Y 306.45,Z 331.601,A -85,B 0,C 180,E1 -16675.646,E2 -16675.646} C_VEL
LIN {X 0,Y 306.362,Z 321.034,A -85,B 0,C 180,E1 -16677.511,E2 -16677.511} C_VEL
LIN {X 0,Y 304.997,Z 309.831,A -85,B 0,C 180,E1 -16679.622,E2 -16679.622} C_VEL
LIN {X 0,Y 303.024,Z 300.08,A -85,B 0,C 180,E1 -16681.647,E2 -16681.647} C_VEL
LIN {X 0,Y 300.096,Z 289.606,A -85,B 0,C 180,E1 -16684.199,E2 -16684.199} C_VEL
LIN {X 0,Y 298.68,Z 285.543,A -85,B 0,C 180,E1 -16685.401,E2 -16685.401} C_VEL
LIN {X 0,Y 298.365,Z 283.868,A -85,B 0,C 180,E1 -16685.812,E2 -16685.812} C_VEL
LIN {X 0,Y 296.393,Z 280.118,A -85,B 0,C 180,E1 -16687.408,E2 -16687.408} C_VEL
LIN {X 0,Y 295.338,Z 276.19,A -85,B 0,C 180,E1 -16688.875,E2 -16688.875} C_VEL
LIN {X 0,Y 295.217,Z 274.039,A -85,B 0,C 180,E1 -16691.804,E2 -16691.804} C_VEL
LIN {X 0,Y 294.89,Z 271.898,A -85,B 0,C 180,E1 -16695.642,E2 -16695.642} C_VEL
LIN {X 0,Y 294.651,Z 270.89,A -85,B 0,C 180,E1 -16698.098,E2 -16698.098} C_VEL
LIN {X 0,Y 294.364,Z 269.944,A -85,B 0,C 180,E1 -16701.697,E2 -16701.697} C_VEL
LIN {X 0,Y 296.074,Z 273.033,A -85,B 0,C 180,E1 -16703.811,E2 -16703.811} C_VEL
LIN {X 0,Y 297.423,Z 274.021,A -85,B 0,C 180,E1 -16704.851,E2 -16704.851} C_VEL
LIN {X 0,Y 301.148,Z 280.038,A -85,B 0,C 180,E1 -16707.779,E2 -16707.779} C_VEL
LIN {X 0,Y 303.356,Z 284.224,A -85,B 0,C 180,E1 -16709.357,E2 -16709.357} C_VEL
LIN {X 0,Y 305.139,Z 287.836,A -85,B 0,C 180,E1 -16710.582,E2 -16710.582} C_VEL
LIN {X 0,Y 308.332,Z 295.693,A -85,B 0,C 180,E1 -16712.879,E2 -16712.879} C_VEL
LIN {X 0,Y 310.774,Z 304.889,A -85,B 0,C 180,E1 -16715.16,E2 -16715.16} C_VEL
LIN {X 0,Y 311.375,Z 309.636,A -85,B 0,C 180,E1 -16716.217,E2 -16716.217} C_VEL
LIN {X 0,Y 308.08,Z 320.259,A -85,B 0,C 180,E1 -16717.889,E2 -16717.889} C_VEL
LIN {X 0,Y 304.682,Z 329.97,A -85,B 0,C 180,E1 -16719.757,E2 -16719.757} C_VEL
LIN {X 0,Y 301.739,Z 337.913,A -85,B 0,C 180,E1 -16721.673,E2 -16721.673} C_VEL
LIN {X 0,Y 299.109,Z 344.498,A -85,B 0,C 180,E1 -16723.623,E2 -16723.623} C_VEL
LIN {X 0,Y 296.842,Z 349.886,A -85,B 0,C 180,E1 -16725.606,E2 -16725.606} C_VEL
LIN {X 0,Y 294.725,Z 354.681,A -85,B 0,C 180,E1 -16727.876,E2 -16727.876} C_VEL
LIN {X 0,Y 292.744,Z 358.481,A -85,B 0,C 180,E1 -16730.326,E2 -16730.326} C_VEL
LIN {X 0,Y 291.593,Z 361.027,A -85,B 0,C 180,E1 -16733.079,E2 -16733.079} C_VEL
LIN {X 0,Y 290.724,Z 362.101,A -85,B 0,C 180,E1 -16735.841,E2 -16735.841} C_VEL
LIN {X 0,Y 290.251,Z 362.048,A -85,B 0,C 180,E1 -16737.224,E2 -16737.224} C_VEL
LIN {X 0,Y 289.752,Z 360.742,A -85,B 0,C 180,E1 -16740,E2 -16740} C_VEL
LIN {X 0,Y 289.674,Z 359.507,A -85,B 0,C 180,E1 -16741.39,E2 -16741.39} C_VEL
LIN {X 0,Y 289.726,Z 356.837,A -85,B 0,C 180,E1 -16743.477,E2 -16743.477} C_VEL
LIN {X 0,Y 289.813,Z 353.172,A -85,B 0,C 180,E1 -16745.567,E2 -16745.567} C_VEL
LIN {X 0,Y 290.089,Z 348.423,A -85,B 0,C 180,E1 -16747.658,E2 -16747.658} C_VEL
LIN {X 0,Y 290.559,Z 341.289,A -85,B 0,C 180,E1 -16750.1,E2 -16750.1} C_VEL
LIN {X 0,Y 291.14,Z 333.625,A -85,B 0,C 180,E1 -16752.194,E2 -16752.194} C_VEL
LIN {X 0,Y 291.955,Z 325.931,A -85,B 0,C 180,E1 -16753.929,E2 -16753.929} C_VEL
LIN {X 0,Y 292.825,Z 315.709,A -85,B 0,C 180,E1 -16755.834,E2 -16755.834} C_VEL
LIN {X 0,Y 293.867,Z 304.19,A -85,B 0,C 180,E1 -16757.574,E2 -16757.574} C_VEL
LIN {X 0,Y 294.873,Z 292.869,A -85,B 0,C 180,E1 -16758.95,E2 -16758.95} C_VEL
LIN {X 0,Y 295.415,Z 286.63,A -85,B 0,C 180,E1 -16759.591,E2 -16759.591} C_VEL
LIN {X 0,Y 293.15,Z 274.106,A -85,B 0,C 180,E1 -16760.772,E2 -16760.772} C_VEL
LIN {X 0,Y 290.629,Z 260.045,A -85,B 0,C 180,E1 -16761.794,E2 -16761.794} C_VEL
LIN {X 0,Y 289.977,Z 256.267,A -85,B 0,C 180,E1 -16762.021,E2 -16762.021} C_VEL
LIN {X 0,Y 290.138,Z 252.416,A -85,B 0,C 180,E1 -16766.329,E2 -16766.329} C_VEL
LIN {X 0,Y 290.562,Z 252.289,A -85,B 0,C 180,E1 -16770.527,E2 -16770.527} C_VEL
LIN {X 0,Y 290.983,Z 252.237,A -85,B 0,C 180,E1 -16773.746,E2 -16773.746} C_VEL
LIN {X 0,Y 291.313,Z 252.2,A -85,B 0,C 180,E1 -16777.237,E2 -16777.237} C_VEL
LIN {X 0,Y 291.335,Z 252.193,A -85,B 0,C 180,E1 -16780.643,E2 -16780.643} C_VEL
LIN {X 0,Y 291.293,Z 252.199,A -85,B 0,C 180,E1 -16784.402,E2 -16784.402} C_VEL
LIN {X 0,Y 291.298,Z 252.198,A -85,B 0,C 180,E1 -16788.411,E2 -16788.411} C_VEL
LIN {X 0,Y 291.337,Z 252.195,A -85,B 0,C 180,E1 -16791.155,E2 -16791.155} C_VEL
LIN {X 0,Y 291.358,Z 252.193,A -85,B 0,C 180,E1 -16794.625,E2 -16794.625} C_VEL
LIN {X 0,Y 291.369,Z 252.189,A -85,B 0,C 180,E1 -16797.95,E2 -16797.95} C_VEL
LIN {X 0,Y 291.358,Z 252.191,A -85,B 0,C 180,E1 -16801.155,E2 -16801.155} C_VEL
LIN {X 0,Y 291.38,Z 252.19,A -85,B 0,C 180,E1 -16804.268,E2 -16804.268} C_VEL
LIN {X 0,Y 291.376,Z 252.187,A -85,B 0,C 180,E1 -16807.299,E2 -16807.299} C_VEL
LIN {X 0,Y 291.461,Z 252.181,A -85,B 0,C 180,E1 -16810.27,E2 -16810.27} C_VEL
LIN {X 0,Y 291.559,Z 252.166,A -85,B 0,C 180,E1 -16814.624,E2 -16814.624} C_VEL
LIN {X 0,Y 291.532,Z 252.169,A -85,B 0,C 180,E1 -16818.88,E2 -16818.88} C_VEL
LIN {X 0,Y 291.654,Z 252.156,A -85,B 0,C 180,E1 -16821.687,E2 -16821.687} C_VEL
LIN {X 0,Y 291.597,Z 252.161,A -85,B 0,C 180,E1 -16824.467,E2 -16824.467} C_VEL
LIN {X 0,Y 291.878,Z 252.126,A -85,B 0,C 180,E1 -16828.62,E2 -16828.62} C_VEL
LIN {X 0,Y 291.873,Z 252.13,A -85,B 0,C 180,E1 -16831.38,E2 -16831.38} C_VEL
LIN {X 0,Y 291.638,Z 252.244,A -85,B 0,C 180,E1 -16833.281,E2 -16833.281} C_VEL
LIN {X 0,Y 291.835,Z 257.324,A -85,B 0,C 180,E1 -16836.221,E2 -16836.221} C_VEL
LIN {X 0,Y 291.426,Z 264.661,A -85,B 0,C 180,E1 -16840.42,E2 -16840.42} C_VEL
LIN {X 0,Y 291.169,Z 270.898,A -85,B 0,C 180,E1 -16843.967,E2 -16843.967} C_VEL
LIN {X 0,Y 290.941,Z 277.223,A -85,B 0,C 180,E1 -16847.575,E2 -16847.575} C_VEL
LIN {X 0,Y 290.874,Z 279.32,A -85,B 0,C 180,E1 -16848.67,E2 -16848.67} C_VEL
LIN {X 0,Y 292.689,Z 289.084,A -85,B 0,C 180,E1 -16849.267,E2 -16849.267} C_VEL
LIN {X 0,Y 294.151,Z 297.614,A -85,B 0,C 180,E1 -16849.951,E2 -16849.951} C_VEL
LIN {X 0,Y 295.118,Z 305.774,A -85,B 0,C 180,E1 -16850.747,E2 -16850.747} C_VEL
LIN {X 0,Y 294.291,Z 316.301,A -85,B 0,C 180,E1 -16851.932,E2 -16851.932} C_VEL
LIN {X 0,Y 293.358,Z 325.409,A -85,B 0,C 180,E1 -16853.284,E2 -16853.284} C_VEL
LIN {X 0,Y 292.723,Z 331.832,A -85,B 0,C 180,E1 -16854.448,E2 -16854.448} C_VEL
LIN {X 0,Y 291.871,Z 339.095,A -85,B 0,C 180,E1 -16856.058,E2 -16856.058} C_VEL
LIN {X 0,Y 291.188,Z 345.017,A -85,B 0,C 180,E1 -16857.685,E2 -16857.685} C_VEL
LIN {X 0,Y 290.586,Z 350.183,A -85,B 0,C 180,E1 -16859.461,E2 -16859.461} C_VEL
LIN {X 0,Y 290.128,Z 354.233,A -85,B 0,C 180,E1 -16861.268,E2 -16861.268} C_VEL
LIN {X 0,Y 289.807,Z 357.196,A -85,B 0,C 180,E1 -16863.068,E2 -16863.068} C_VEL
LIN {X 0,Y 289.621,Z 358.785,A -85,B 0,C 180,E1 -16864.406,E2 -16864.406} C_VEL
LIN {X 0,Y 289.456,Z 360.396,A -85,B 0,C 180,E1 -16866.751,E2 -16866.751} C_VEL
LIN {X 0,Y 289.618,Z 360.563,A -85,B 0,C 180,E1 -16869.119,E2 -16869.119} C_VEL
LIN {X 0,Y 289.997,Z 359.493,A -85,B 0,C 180,E1 -16871.298,E2 -16871.298} C_VEL
LIN {X 0,Y 290.596,Z 357.099,A -85,B 0,C 180,E1 -16873.485,E2 -16873.485} C_VEL
LIN {X 0,Y 291.325,Z 353.403,A -85,B 0,C 180,E1 -16875.604,E2 -16875.604} C_VEL
LIN {X 0,Y 292.296,Z 348.404,A -85,B 0,C 180,E1 -16877.682,E2 -16877.682} C_VEL
LIN {X 0,Y 293.546,Z 341.794,A -85,B 0,C 180,E1 -16879.727,E2 -16879.727} C_VEL
LIN {X 0,Y 294.753,Z 335.13,A -85,B 0,C 180,E1 -16881.312,E2 -16881.312} C_VEL
LIN {X 0,Y 295.951,Z 327.9,A -85,B 0,C 180,E1 -16882.705,E2 -16882.705} C_VEL
LIN {X 0,Y 297.218,Z 319.052,A -85,B 0,C 180,E1 -16884.083,E2 -16884.083} C_VEL
LIN {X 0,Y 298.305,Z 310.3,A -85,B 0,C 180,E1 -16885.157,E2 -16885.157} C_VEL
LIN {X 0,Y 296.861,Z 299.878,A -85,B 0,C 180,E1 -16886.339,E2 -16886.339} C_VEL
LIN {X 0,Y 294.781,Z 290.682,A -85,B 0,C 180,E1 -16887.241,E2 -16887.241} C_VEL
LIN {X 0,Y 291.878,Z 280.485,A -85,B 0,C 180,E1 -16888.114,E2 -16888.114} C_VEL
LIN {X 0,Y 292.253,Z 273.744,A -85,B 0,C 180,E1 -16892.036,E2 -16892.036} C_VEL
LIN {X 0,Y 292.752,Z 265.8,A -85,B 0,C 180,E1 -16896.664,E2 -16896.664} C_VEL
LIN {X 0,Y 292.957,Z 261.239,A -85,B 0,C 180,E1 -16899.326,E2 -16899.326} C_VEL
LIN {X 0,Y 292.296,Z 256.215,A -85,B 0,C 180,E1 -16902.509,E2 -16902.509} C_VEL
LIN {X 0,Y 291.573,Z 252.165,A -85,B 0,C 180,E1 -16905.088,E2 -16905.088} C_VEL
LIN {X 0,Y 291.538,Z 252.174,A -85,B 0,C 180,E1 -16908.88,E2 -16908.88} C_VEL
LIN {X 0,Y 291.557,Z 252.17,A -85,B 0,C 180,E1 -16910.026,E2 -16910.026} C_VEL
LIN {X 0,Y 291.274,Z 252.208,A -85,B 0,C 180,E1 -16910.798,E2 -16910.798} C_VEL
LIN {X 0,Y 289.313,Z 252.454,A -85,B 0,C 180,E1 -16912.311,E2 -16912.311} C_VEL
LIN {X 0,Y 285.555,Z 252.917,A -85,B 0,C 180,E1 -16914.582,E2 -16914.582} C_VEL
LIN {X 0,Y 284.587,Z 253.035,A -85,B 0,C 180,E1 -16915.766,E2 -16915.766} C_VEL
LIN {X 0,Y 284.554,Z 253.037,A -85,B 0,C 180,E1 -16916.166,E2 -16916.166} C_VEL
LIN {X 0,Y 284.856,Z 253.004,A -85,B 0,C 180,E1 -16918.586,E2 -16918.586} C_VEL
LIN {X 0,Y 284.856,Z 253.001,A -85,B 0,C 180,E1 -16921.414,E2 -16921.414} C_VEL
LIN {X 0,Y 284.655,Z 253.029,A -85,B 0,C 180,E1 -16927.091,E2 -16927.091} C_VEL
LIN {X 0,Y 284.519,Z 253.045,A -85,B 0,C 180,E1 -16929.957,E2 -16929.957} C_VEL
LIN {X 0,Y 284.483,Z 253.048,A -85,B 0,C 180,E1 -16934.303,E2 -16934.303} C_VEL
LIN {X 0,Y 284.427,Z 253.056,A -85,B 0,C 180,E1 -16937.248,E2 -16937.248} C_VEL
LIN {X 0,Y 284.378,Z 253.063,A -85,B 0,C 180,E1 -16940.242,E2 -16940.242} C_VEL
LIN {X 0,Y 284.34,Z 253.066,A -85,B 0,C 180,E1 -16944.846,E2 -16944.846} C_VEL
LIN {X 0,Y 284.333,Z 253.068,A -85,B 0,C 180,E1 -16948.01,E2 -16948.01} C_VEL
LIN {X 0,Y 284.297,Z 253.071,A -85,B 0,C 180,E1 -16951.274,E2 -16951.274} C_VEL
LIN {X 0,Y 284.342,Z 253.065,A -85,B 0,C 180,E1 -16955.348,E2 -16955.348} C_VEL
LIN {X 0,Y 284.32,Z 253.069,A -85,B 0,C 180,E1 -16958.168,E2 -16958.168} C_VEL
LIN {X 0,Y 284.283,Z 253.071,A -85,B 0,C 180,E1 -16962.127,E2 -16962.127} C_VEL
LIN {X 0,Y 284.424,Z 253.233,A -85,B 0,C 180,E1 -16964.504,E2 -16964.504} C_VEL
LIN {X 0,Y 285.331,Z 258.2,A -85,B 0,C 180,E1 -16968.315,E2 -16968.315} C_VEL
LIN {X 0,Y 286.156,Z 263.392,A -85,B 0,C 180,E1 -16972.121,E2 -16972.121} C_VEL
LIN {X 0,Y 286.27,Z 266.206,A -85,B 0,C 180,E1 -16974.112,E2 -16974.112} C_VEL
LIN {X 0,Y 285.491,Z 270.774,A -85,B 0,C 180,E1 -16977.209,E2 -16977.209} C_VEL
LIN {X 0,Y 284.524,Z 276.744,A -85,B 0,C 180,E1 -16981.206,E2 -16981.206} C_VEL
LIN {X 0,Y 283.784,Z 282.698,A -85,B 0,C 180,E1 -16985.053,E2 -16985.053} C_VEL
LIN {X 0,Y 285.077,Z 296.527,A -85,B 0,C 180,E1 -16987.726,E2 -16987.726} C_VEL
LIN {X 0,Y 285.215,Z 299.598,A -85,B 0,C 180,E1 -16988.261,E2 -16988.261} C_VEL
LIN {X 0,Y 287.082,Z 314.916,A -85,B 0,C 180,E1 -16989.076,E2 -16989.076} C_VEL
LIN {X 0,Y 288.103,Z 325.504,A -85,B 0,C 180,E1 -16989.902,E2 -16989.902} C_VEL
LIN {X 0,Y 288.637,Z 332.998,A -85,B 0,C 180,E1 -16990.625,E2 -16990.625} C_VEL
LIN {X 0,Y 287.942,Z 341.274,A -85,B 0,C 180,E1 -16991.5,E2 -16991.5} C_VEL
LIN {X 0,Y 287.059,Z 349.314,A -85,B 0,C 180,E1 -16992.548,E2 -16992.548} C_VEL
LIN {X 0,Y 286.109,Z 356.373,A -85,B 0,C 180,E1 -16993.659,E2 -16993.659} C_VEL
LIN {X 0,Y 285.266,Z 363.399,A -85,B 0,C 180,E1 -16995.008,E2 -16995.008} C_VEL
LIN {X 0,Y 284.484,Z 369.531,A -85,B 0,C 180,E1 -16996.427,E2 -16996.427} C_VEL
LIN {X 0,Y 283.619,Z 375.826,A -85,B 0,C 180,E1 -16998.204,E2 -16998.204} C_VEL
LIN {X 0,Y 283.099,Z 380.849,A -85,B 0,C 180,E1 -16999.993,E2 -16999.993} C_VEL
LIN {X 0,Y 282.709,Z 385.378,A -85,B 0,C 180,E1 -17002.142,E2 -17002.142} C_VEL
LIN {X 0,Y 282.542,Z 388.564,A -85,B 0,C 180,E1 -17004.29,E2 -17004.29} C_VEL
LIN {X 0,Y 282.507,Z 390.043,A -85,B 0,C 180,E1 -17005.72,E2 -17005.72} C_VEL
LIN {X 0,Y 282.58,Z 391.025,A -85,B 0,C 180,E1 -17007.149,E2 -17007.149} C_VEL
LIN {X 0,Y 282.64,Z 391.424,A -85,B 0,C 180,E1 -17008.575,E2 -17008.575} C_VEL
LIN {X 0,Y 282.787,Z 391.281,A -85,B 0,C 180,E1 -17010,E2 -17010} C_VEL
LIN {X 0,Y 282.707,Z 391.324,A -85,B 0,C 180,E1 -17011.425,E2 -17011.425} C_VEL
LIN {X 0,Y 282.437,Z 391.837,A -85,B 0,C 180,E1 -17014.281,E2 -17014.281} C_VEL
LIN {X 0,Y 282.408,Z 391.503,A -85,B 0,C 180,E1 -17015.713,E2 -17015.713} C_VEL
LIN {X 0,Y 282.781,Z 389.613,A -85,B 0,C 180,E1 -17018.576,E2 -17018.576} C_VEL
LIN {X 0,Y 283.706,Z 386.199,A -85,B 0,C 180,E1 -17021.431,E2 -17021.431} C_VEL
LIN {X 0,Y 284.824,Z 382.565,A -85,B 0,C 180,E1 -17023.557,E2 -17023.557} C_VEL
LIN {X 0,Y 286.634,Z 377.974,A -85,B 0,C 180,E1 -17025.647,E2 -17025.647} C_VEL
LIN {X 0,Y 288.829,Z 371.374,A -85,B 0,C 180,E1 -17028.074,E2 -17028.074} C_VEL
LIN {X 0,Y 291.866,Z 363.138,A -85,B 0,C 180,E1 -17030.436,E2 -17030.436} C_VEL
LIN {X 0,Y 295.696,Z 353.061,A -85,B 0,C 180,E1 -17032.72,E2 -17032.72} C_VEL
LIN {X 0,Y 299.19,Z 342.639,A -85,B 0,C 180,E1 -17034.643,E2 -17034.643} C_VEL
LIN {X 0,Y 300.439,Z 335.171,A -85,B 0,C 180,E1 -17036.016,E2 -17036.016} C_VEL
LIN {X 0,Y 300.817,Z 325.407,A -85,B 0,C 180,E1 -17037.857,E2 -17037.857} C_VEL
LIN {X 0,Y 300.071,Z 314.988,A -85,B 0,C 180,E1 -17039.936,E2 -17039.936} C_VEL
LIN {X 0,Y 298.839,Z 307.441,A -85,B 0,C 180,E1 -17041.592,E2 -17041.592} C_VEL
LIN {X 0,Y 297.327,Z 299.503,A -85,B 0,C 180,E1 -17043.478,E2 -17043.478} C_VEL
LIN {X 0,Y 296.196,Z 294.913,A -85,B 0,C 180,E1 -17044.713,E2 -17044.713} C_VEL
LIN {X 0,Y 295.051,Z 291.029,A -85,B 0,C 180,E1 -17045.917,E2 -17045.917} C_VEL
LIN {X 0,Y 294.798,Z 289.5,A -85,B 0,C 180,E1 -17046.336,E2 -17046.336} C_VEL
LIN {X 0,Y 292.888,Z 284.887,A -85,B 0,C 180,E1 -17048.305,E2 -17048.305} C_VEL
LIN {X 0,Y 292.381,Z 282.444,A -85,B 0,C 180,E1 -17049.211,E2 -17049.211} C_VEL
LIN {X 0,Y 289.947,Z 278.34,A -85,B 0,C 180,E1 -17052.742,E2 -17052.742} C_VEL
LIN {X 0,Y 289.349,Z 276.543,A -85,B 0,C 180,E1 -17055.22,E2 -17055.22} C_VEL
LIN {X 0,Y 289.452,Z 275.972,A -85,B 0,C 180,E1 -17057.168,E2 -17057.168} C_VEL
LIN {X 0,Y 290.978,Z 276.357,A -85,B 0,C 180,E1 -17060.616,E2 -17060.616} C_VEL
LIN {X 0,Y 291.415,Z 276.472,A -85,B 0,C 180,E1 -17061.168,E2 -17061.168} C_VEL
LIN {X 0,Y 292.737,Z 278.822,A -85,B 0,C 180,E1 -17063.116,E2 -17063.116} C_VEL
LIN {X 0,Y 294.832,Z 281.226,A -85,B 0,C 180,E1 -17065.104,E2 -17065.104} C_VEL
LIN {X 0,Y 297.453,Z 285.815,A -85,B 0,C 180,E1 -17067.426,E2 -17067.426} C_VEL
LIN {X 0,Y 300.498,Z 292.197,A -85,B 0,C 180,E1 -17069.924,E2 -17069.924} C_VEL
LIN {X 0,Y 303.336,Z 300.086,A -85,B 0,C 180,E1 -17072.395,E2 -17072.395} C_VEL
LIN {X 0,Y 305.206,Z 307.988,A -85,B 0,C 180,E1 -17074.515,E2 -17074.515} C_VEL
LIN {X 0,Y 305.736,Z 312.227,A -85,B 0,C 180,E1 -17075.558,E2 -17075.558} C_VEL
LIN {X 0,Y 301.904,Z 323.376,A -85,B 0,C 180,E1 -17077.412,E2 -17077.412} C_VEL
LIN {X 0,Y 298.38,Z 332.508,A -85,B 0,C 180,E1 -17079.31,E2 -17079.31} C_VEL
LIN {X 0,Y 294.787,Z 341.234,A -85,B 0,C 180,E1 -17081.585,E2 -17081.585} C_VEL
LIN {X 0,Y 291.687,Z 348.158,A -85,B 0,C 180,E1 -17083.914,E2 -17083.914} C_VEL
LIN {X 0,Y 289.388,Z 352.917,A -85,B 0,C 180,E1 -17085.945,E2 -17085.945} C_VEL
LIN {X 0,Y 287.54,Z 356.656,A -85,B 0,C 180,E1 -17088.009,E2 -17088.009} C_VEL
LIN {X 0,Y 285.818,Z 359.49,A -85,B 0,C 180,E1 -17090.089,E2 -17090.089} C_VEL
LIN {X 0,Y 284.609,Z 361.807,A -85,B 0,C 180,E1 -17092.908,E2 -17092.908} C_VEL
LIN {X 0,Y 284.075,Z 362.42,A -85,B 0,C 180,E1 -17094.321,E2 -17094.321} C_VEL
LIN {X 0,Y 283.67,Z 362.617,A -85,B 0,C 180,E1 -17095.738,E2 -17095.738} C_VEL
